KUKA KRL program: MyProgram_203().src

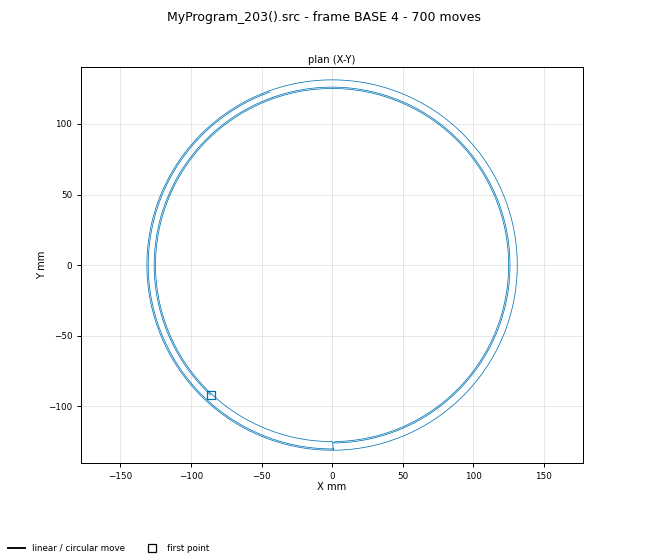
[picture p0: tool path of MyProgram_203().src in frame BASE 4, 700 of 700 moves have a stored position in this frame; points joined in program order, loops and branches not executed]
&ACCESS RVP
&REL 1
&PARAM TEMPLATE = C:\KRC\Roboter\Template\vorgabe
&PARAM EDITMASK = *
DEF MyProgram_203()
; ---- Setting reference (Base) ----
$BASE = BASE_DATA[4]

; --------------------------
; ---- Setting tool (TCP) ----
$TOOL = TOOL_DATA[3]
; --------------------------

$VEL.CP = VEL_APROX_PRINT
Startdeposition()
$VEL.CP = VEL_PRINT
LIN {X -86.0761,Y -92.1467,Z 145,A -135.8963,B 21.9718,C -0.8867,E1 21.8788,E2 583.2193} C_DIS
LIN {X -89.1832,Y -89.1435,Z 145,A -137.9047,B 21.9718,C -0.889,E1 21.8748,E2 585.2313} C_DIS
LIN {X -92.1675,Y -86.0537,Z 145,A -139.8494,B 21.9716,C -0.8935,E1 21.871,E2 587.1736} C_DIS
LIN {X -95.1424,Y -82.7529,Z 145,A -141.8562,B 21.9714,C -0.8986,E1 21.8673,E2 589.1772} C_DIS
LIN {X -97.9193,Y -79.4482,Z 145,A -144.0903,B 21.9716,C -0.8923,E1 21.8633,E2 591.4401} C_DIS
LIN {X -99.986,Y -76.8307,Z 145,A -145.2029,B 21.9709,C -0.9119,E1 21.8615,E2 592.506} C_DIS
LIN {X -101.9983,Y -74.1381,Z 145,A -146.8853,B 21.9709,C -0.9095,E1 21.8587,E2 594.2043} C_DIS
LIN {X -104.8548,Y -70.0396,Z 145,A -149.0462,B 21.9706,C -0.9196,E1 21.8553,E2 596.3505} C_DIS
LIN {X -106.8541,Y -66.9509,Z 145,A -150.8688,B 21.9706,C -0.9179,E1 21.8525,E2 598.1883} C_DIS
LIN {X -109.0384,Y -63.3304,Z 145,A -153.5164,B 21.9715,C -0.8945,E1 21.8487,E2 600.9146} C_DIS
LIN {X -111.7045,Y -58.4954,Z 145,A -154.9531,B 21.9696,C -0.9434,E1 21.847,E2 602.2285} C_DIS
LIN {X -113.7032,Y -54.5088,Z 145,A -157.2159,B 21.9697,C -0.9397,E1 21.8441,E2 604.5155} C_DIS
LIN {X -115.0389,Y -51.6302,Z 145,A -158.7729,B 21.9697,C -0.9392,E1 21.8423,E2 606.0836} C_DIS
LIN {X -116.4531,Y -48.3564,Z 145,A -160.379,B 21.9696,C -0.9444,E1 21.8405,E2 607.686} C_DIS
LIN {X -117.9838,Y -44.4918,Z 145,A -162.2933,B 21.9694,C -0.9489,E1 21.8386,E2 609.6006} C_DIS
LIN {X -119.2139,Y -41.082,Z 145,A -163.8822,B 21.9691,C -0.956,E1 21.8371,E2 611.1808} C_DIS
LIN {X -120.4558,Y -37.2854,Z 145,A -165.5654,B 21.9686,C -0.9666,E1 21.8357,E2 612.8467} C_DIS
LIN {X -121.1863,Y -34.8412,Z 145,A -167.1929,B 21.9692,C -0.9518,E1 21.8344,E2 614.525} C_DIS
LIN {X -122.4757,Y -29.9927,Z 145,A -169.1331,B 21.9684,C -0.9719,E1 21.8331,E2 616.424} C_DIS
LIN {X -123.2253,Y -26.7432,Z 145,A -170.7725,B 21.9684,C -0.9718,E1 21.8321,E2 618.0751} C_DIS
LIN {X -123.9753,Y -23.0268,Z 145,A -172.5489,B 21.9683,C -0.975,E1 21.8311,E2 619.8549} C_DIS
LIN {X -124.6142,Y -19.261,Z 145,A -174.2077,B 21.9679,C -0.9834,E1 21.8304,E2 621.5024} C_DIS
LIN {X -125.1352,Y -15.5323,Z 145,A -176.0548,B 21.9679,C -0.9834,E1 21.8297,E2 623.3622} C_DIS
LIN {X -125.5578,Y -11.6249,Z 145,A -177.7788,B 21.9676,C -0.9915,E1 21.8292,E2 625.0765} C_DIS
LIN {X -125.8536,Y -7.7849,Z 145,A -179.5233,B 21.9673,C -0.9973,E1 21.8289,E2 626.8176} C_DIS
LIN {X -126.0388,Y -3.7439,Z 145,A 178.611,B 21.9671,C -1.002,E1 21.8287,E2 628.6834} C_DIS
LIN {X -126.0974,Y -0.0263,Z 145,A 176.8014,B 21.9671,C -1.0027,E1 21.8287,E2 630.5039} C_DIS
LIN {X -126.0368,Y 3.817,Z 145,A 175.0886,B 21.9668,C -1.0096,E1 21.8287,E2 632.2099} C_DIS
LIN {X -125.8518,Y 7.8139,Z 145,A 173.3197,B 21.9665,C -1.0173,E1 21.829,E2 633.9703} C_DIS
LIN {X -125.5347,Y 11.8647,Z 145,A 171.4401,B 21.9663,C -1.0219,E1 21.8295,E2 635.8506} C_DIS
LIN {X -125.1188,Y 15.6685,Z 145,A 169.6388,B 21.9661,C -1.025,E1 21.83,E2 637.6561} C_DIS
LIN {X -124.595,Y 19.3851,Z 145,A 168.0151,B 21.9657,C -1.0337,E1 21.8307,E2 639.2677} C_DIS
LIN {X -123.9237,Y 23.2965,Z 145,A 165.8228,B 21.9661,C -1.0243,E1 21.8318,E2 641.5001} C_DIS
LIN {X -123.2397,Y 26.6765,Z 145,A 164.7208,B 21.9651,C -1.0473,E1 21.8324,E2 642.5479} C_DIS
LIN {X -122.5731,Y 29.5888,Z 145,A 163.2246,B 21.9651,C -1.0462,E1 21.8334,E2 644.0573} C_DIS
LIN {X -121.6224,Y 33.2883,Z 145,A 161.4104,B 21.9651,C -1.0485,E1 21.8347,E2 645.8773} C_DIS
LIN {X -120.307,Y 37.7657,Z 145,A 159.4485,B 21.9645,C -1.0613,E1 21.8363,E2 647.818} C_DIS
LIN {X -119.4002,Y 40.5435,Z 145,A 158.0205,B 21.9645,C -1.0614,E1 21.8375,E2 649.2549} C_DIS
LIN {X -118.558,Y 42.9378,Z 145,A 156.8422,B 21.9644,C -1.064,E1 21.8386,E2 650.434} C_DIS
LIN {X -117.1974,Y 46.5278,Z 145,A 155.0158,B 21.9643,C -1.0661,E1 21.8405,E2 652.2666} C_DIS
LIN {X -113.3052,Y 55.3334,Z 145,A 150.8392,B 21.9633,C -1.0868,E1 21.8452,E2 656.4139} C_DIS
LIN {X -110.7395,Y 60.3063,Z 145,A 148.2402,B 21.963,C -1.092,E1 21.8486,E2 659.0152} C_DIS
LIN {X -108.9465,Y 63.4891,Z 145,A 146.3727,B 21.9632,C -1.0886,E1 21.8512,E2 660.903} C_DIS
LIN {X -106.7944,Y 67.0458,Z 145,A 144.4384,B 21.963,C -1.0921,E1 21.854,E2 662.8392} C_DIS
LIN {X -104.4846,Y 70.5907,Z 145,A 142.5355,B 21.9628,C -1.0982,E1 21.857,E2 664.7368} C_DIS
LIN {X -102.1644,Y 73.9089,Z 145,A 140.7167,B 21.9625,C -1.104,E1 21.8599,E2 666.5503} C_DIS
LIN {X -99.4483,Y 77.5257,Z 145,A 138.8921,B 21.9618,C -1.1185,E1 21.8629,E2 668.3461} C_DIS
LIN {X -97.8225,Y 79.5671,Z 145,A 137.4168,B 21.9622,C -1.1101,E1 21.8656,E2 669.8517} C_DIS
LIN {X -95.19,Y 82.6983,Z 145,A 135.5368,B 21.962,C -1.114,E1 21.869,E2 671.7312} C_DIS
LIN {X -92.105,Y 86.1209,Z 145,A 133.453,B 21.9617,C -1.1196,E1 21.8729,E2 673.8107} C_DIS
LIN {X -89.2767,Y 89.0495,Z 145,A 131.5891,B 21.9615,C -1.1235,E1 21.8765,E2 675.6733} C_DIS
LIN {X -86.2214,Y 92.0114,Z 145,A 129.6757,B 21.9613,C -1.1287,E1 21.8804,E2 677.5817} C_DIS
LIN {X -83.1134,Y 94.8278,Z 145,A 127.8773,B 21.9609,C -1.1373,E1 21.8841,E2 679.3654} C_DIS
LIN {X -80.3032,Y 97.2188,Z 145,A 126.0625,B 21.9609,C -1.1355,E1 21.888,E2 681.1931} C_DIS
LIN {X -77.0858,Y 99.7893,Z 145,A 124.1693,B 21.9609,C -1.1385,E1 21.8922,E2 683.0862} C_DIS
LIN {X -73.9124,Y 102.1618,Z 145,A 122.2451,B 21.9609,C -1.1373,E1 21.8965,E2 685.0216} C_DIS
LIN {X -70.7167,Y 104.3994,Z 145,A 120.5946,B 21.9605,C -1.1456,E1 21.9003,E2 686.6563} C_DIS
LIN {X -67.5028,Y 106.5059,Z 145,A 118.788,B 21.9605,C -1.1464,E1 21.9045,E2 688.4673} C_DIS
LIN {X -63.9081,Y 108.7007,Z 145,A 116.9174,B 21.9602,C -1.1515,E1 21.909,E2 690.3307} C_DIS
LIN {X -60.038,Y 110.8858,Z 145,A 114.855,B 21.9601,C -1.1532,E1 21.9141,E2 692.3955} C_DIS
LIN {X -56.8206,Y 112.5664,Z 145,A 113.1703,B 21.9601,C -1.1545,E1 21.9182,E2 694.0821} C_DIS
LIN {X -53.2771,Y 114.2861,Z 145,A 111.4983,B 21.9596,C -1.1619,E1 21.9224,E2 695.739} C_DIS
LIN {X -50.183,Y 115.6776,Z 145,A 109.9447,B 21.9596,C -1.1637,E1 21.9264,E2 697.2922} C_DIS
LIN {X -46.4167,Y 117.242,Z 145,A 107.7691,B 21.9601,C -1.1531,E1 21.9321,E2 699.5017} C_DIS
LIN {X -43.3787,Y 118.3991,Z 145,A 106.5136,B 21.9595,C -1.164,E1 21.9353,E2 700.7311} C_DIS
LIN {X -36.9762,Y 120.5504,Z 145,A 103.4705,B 21.9593,C -1.1686,E1 21.9434,E2 703.7683} C_DIS
LIN {X -33.2234,Y 121.6402,Z 145,A 101.5654,B 21.9595,C -1.1651,E1 21.9485,E2 705.6862} C_DIS
LIN {X -29.0003,Y 122.7149,Z 145,A 99.7308,B 21.9591,C -1.1728,E1 21.9535,E2 707.5029} C_DIS
LIN {X -25.2822,Y 123.5334,Z 145,A 98.0319,B 21.9589,C -1.1756,E1 21.9581,E2 709.1969} C_DIS
LIN {X -21.8299,Y 124.1905,Z 145,A 96.3146,B 21.9591,C -1.1718,E1 21.9629,E2 710.9264} C_DIS
LIN {X -17.8466,Y 124.8246,Z 145,A 94.5969,B 21.9588,C -1.1777,E1 21.9676,E2 712.6299} C_DIS
LIN {X -14.2799,Y 125.2846,Z 145,A 92.9165,B 21.9588,C -1.1767,E1 21.9722,E2 714.3144} C_DIS
LIN {X -10.3602,Y 125.668,Z 145,A 91.0232,B 21.9591,C -1.1732,E1 21.9775,E2 716.2181} C_DIS
LIN {X -5.674,Y 125.968,Z 145,A 88.9107,B 21.959,C -1.1748,E1 21.9834,E2 718.327} C_DIS
LIN {X -1.8806,Y 126.0803,Z 145,A 87.2175,B 21.9589,C -1.1765,E1 21.9881,E2 720.0158} C_DIS
LIN {X 2.6511,Y 126.0675,Z 145,A 85.1051,B 21.9589,C -1.1745,E1 21.994,E2 722.1331} C_DIS
LIN {X 6.9515,Y 125.9039,Z 145,A 83.2593,B 21.9588,C -1.1791,E1 21.9991,E2 723.966} C_DIS
LIN {X 10.5423,Y 125.6526,Z 145,A 81.648,B 21.9588,C -1.1801,E1 22.0036,E2 725.5738} C_DIS
LIN {X 14.0573,Y 125.3093,Z 145,A 79.8978,B 21.959,C -1.1736,E1 22.0085,E2 727.3398} C_DIS
LIN {X 18.2331,Y 124.7694,Z 145,A 78.1356,B 21.9587,C -1.1795,E1 22.0133,E2 729.0846} C_DIS
LIN {X 22.0415,Y 124.1527,Z 145,A 76.3822,B 21.9587,C -1.1789,E1 22.0182,E2 730.8376} C_DIS
LIN {X 25.7971,Y 123.4286,Z 145,A 74.5556,B 21.959,C -1.1743,E1 22.0232,E2 732.6739} C_DIS
LIN {X 29.4691,Y 122.6019,Z 145,A 72.9585,B 21.9588,C -1.1782,E1 22.0275,E2 734.2581} C_DIS
LIN {X 32.7186,Y 121.7752,Z 145,A 71.476,B 21.9588,C -1.1789,E1 22.0315,E2 735.7358} C_DIS
LIN {X 36.0284,Y 120.8387,Z 145,A 69.5967,B 21.9595,C -1.1642,E1 22.0366,E2 737.6507} C_DIS
LIN {X 40.2853,Y 119.4862,Z 145,A 67.8211,B 21.9591,C -1.1734,E1 22.0413,E2 739.3978} C_DIS
LIN {X 44.8165,Y 117.8622,Z 145,A 65.6246,B 21.9591,C -1.171,E1 22.047,E2 741.5956} C_DIS
LIN {X 48.3157,Y 116.4701,Z 145,A 63.9039,B 21.9593,C -1.1688,E1 22.0515,E2 743.3176} C_DIS
LIN {X 51.3332,Y 115.1717,Z 145,A 62.4227,B 21.9593,C -1.1676,E1 22.0553,E2 744.7977} C_DIS
LIN {X 54.3914,Y 113.7593,Z 145,A 60.934,B 21.9593,C -1.1676,E1 22.059,E2 746.2821} C_DIS
LIN {X 57.5159,Y 112.2125,Z 145,A 59.2771,B 21.9596,C -1.1624,E1 22.0632,E2 747.9476} C_DIS
LIN {X 61.6301,Y 110.0083,Z 145,A 57.1457,B 21.9598,C -1.159,E1 22.0684,E2 750.0811} C_DIS
LIN {X 65.4184,Y 107.7987,Z 145,A 55.2232,B 21.9598,C -1.159,E1 22.073,E2 751.9964} C_DIS
LIN {X 68.8019,Y 105.6712,Z 145,A 52.7949,B 21.9612,C -1.1295,E1 22.0789,E2 754.4942} C_DIS
LIN {X 72.8559,Y 102.9174,Z 145,A 51.3065,B 21.9598,C -1.158,E1 22.0821,E2 755.9008} C_DIS
LIN {X 75.3902,Y 101.0762,Z 145,A 49.7164,B 21.9603,C -1.1482,E1 22.0857,E2 757.5106} C_DIS
LIN {X 78.8216,Y 98.4244,Z 145,A 47.7508,B 21.9605,C -1.1448,E1 22.09,E2 759.4768} C_DIS
LIN {X 82.0406,Y 95.7576,Z 145,A 45.8388,B 21.9607,C -1.1405,E1 22.0941,E2 761.3916} C_DIS
LIN {X 85.4008,Y 92.7728,Z 145,A 43.8587,B 21.9607,C -1.1392,E1 22.0982,E2 763.3661} C_DIS
LIN {X 88.4403,Y 89.88,Z 145,A 41.9475,B 21.961,C -1.135,E1 22.102,E2 765.2792} C_DIS
LIN {X 91.391,Y 86.8785,Z 145,A 40.0249,B 21.9612,C -1.1304,E1 22.1058,E2 767.2045} C_DIS
LIN {X 93.6073,Y 84.4858,Z 145,A 38.5847,B 21.9612,C -1.1289,E1 22.1085,E2 768.6413} C_DIS
LIN {X 96.3788,Y 81.31,Z 145,A 36.0715,B 21.9628,C -1.0979,E1 22.1132,E2 771.2237} C_DIS
LIN {X 99.535,Y 77.4131,Z 145,A 34.5935,B 21.9613,C -1.1281,E1 22.1156,E2 772.6133} C_DIS
LIN {X 101.1414,Y 75.3027,Z 145,A 33.1546,B 21.962,C -1.1147,E1 22.118,E2 774.0801} C_DIS
LIN {X 103.7943,Y 71.6024,Z 145,A 31.1509,B 21.962,C -1.1124,E1 22.1212,E2 776.0786} C_DIS
LIN {X 106.1382,Y 68.0791,Z 145,A 29.1772,B 21.9624,C -1.1052,E1 22.1242,E2 778.0601} C_DIS
LIN {X 108.4285,Y 64.3692,Z 145,A 27.304,B 21.9624,C -1.1048,E1 22.1269,E2 779.9233} C_DIS
LIN {X 110.3157,Y 61.0781,Z 145,A 25.7873,B 21.9622,C -1.1095,E1 22.129,E2 781.4184} C_DIS
LIN {X 111.6871,Y 58.5286,Z 145,A 24.3527,B 21.9626,C -1.1006,E1 22.1309,E2 782.868} C_DIS
LIN {X 113.193,Y 55.5608,Z 145,A 22.834,B 21.9629,C -1.0961,E1 22.1328,E2 784.3893} C_DIS
LIN {X 114.5601,Y 52.6845,Z 145,A 21.3651,B 21.9631,C -1.091,E1 22.1345,E2 785.8626} C_DIS
LIN {X 117.083,Y 46.8114,Z 145,A 18.5463,B 21.9633,C -1.0865,E1 22.1376,E2 788.6754} C_DIS
LIN {X 118.1916,Y 43.937,Z 145,A 17.1359,B 21.9635,C -1.0819,E1 22.139,E2 790.0889} C_DIS
LIN {X 119.3991,Y 40.5467,Z 145,A 15.2634,B 21.9642,C -1.0663,E1 22.1407,E2 791.9907} C_DIS
LIN {X 120.5527,Y 36.9689,Z 145,A 13.7751,B 21.964,C -1.0712,E1 22.142,E2 793.4562} C_DIS
LIN {X 121.6013,Y 33.3639,Z 145,A 12.0113,B 21.9644,C -1.0634,E1 22.1433,E2 795.2292} C_DIS
LIN {X 122.5655,Y 29.6202,Z 145,A 10.3631,B 21.9644,C -1.063,E1 22.1444,E2 796.8674} C_DIS
LIN {X 123.3293,Y 26.2616,Z 145,A 8.698,B 21.9648,C -1.0536,E1 22.1454,E2 798.5463} C_DIS
LIN {X 124.1128,Y 22.264,Z 145,A 6.9712,B 21.9648,C -1.0536,E1 22.1463,E2 800.2616} C_DIS
LIN {X 124.6972,Y 18.7236,Z 145,A 5.3351,B 21.9651,C -1.0482,E1 22.147,E2 801.9009} C_DIS
LIN {X 125.181,Y 15.1483,Z 145,A 3.697,B 21.9653,C -1.0431,E1 22.1476,E2 803.5414} C_DIS
LIN {X 125.5665,Y 11.5343,Z 145,A 1.8734,B 21.9659,C -1.03,E1 22.1481,E2 805.3873} C_DIS
LIN {X 125.8923,Y 7.1553,Z 145,A -0.0848,B 21.9661,C -1.0253,E1 22.1485,E2 807.3445} C_DIS
LIN {X 126.0698,Y 2.5107,Z 145,A -2.008,B 21.9661,C -1.0272,E1 22.1486,E2 809.2494} C_DIS
LIN {X 126.0934,Y -0.7076,Z 145,A -3.5783,B 21.9664,C -1.0176,E1 22.1486,E2 810.8345} C_DIS
LIN {X 126.0148,Y -4.4933,Z 145,A -4.9898,B 21.9661,C -1.0263,E1 22.1486,E2 812.2131} C_DIS
LIN {X 125.8818,Y -7.3261,Z 145,A -6.4589,B 21.9666,C -1.0139,E1 22.1483,E2 813.7052} C_DIS
LIN {X 125.6288,Y -10.8246,Z 145,A -7.9964,B 21.9667,C -1.0114,E1 22.148,E2 815.2388} C_DIS
LIN {X 125.2804,Y -14.3147,Z 145,A -9.8028,B 21.9674,C -0.9965,E1 22.1474,E2 817.0724} C_DIS
LIN {X 124.5584,Y -19.6216,Z 145,A -11.9587,B 21.9671,C -1.0015,E1 22.1466,E2 819.2004} C_DIS
LIN {X 123.9753,Y -23.0268,Z 145,A -13.6498,B 21.9676,C -0.9909,E1 22.1457,E2 820.9081} C_DIS
LIN {X 123.2202,Y -26.7671,Z 145,A -15.2366,B 21.9676,C -0.9922,E1 22.1448,E2 822.4809} C_DIS
LIN {X 122.5183,Y -29.816,Z 145,A -16.6631,B 21.9678,C -0.9875,E1 22.1439,E2 823.9104} C_DIS
LIN {X 121.587,Y -33.415,Z 145,A -19.208,B 21.9696,C -0.9431,E1 22.142,E2 826.556} C_DIS
LIN {X 119.9115,Y -39.004,Z 145,A -21.2058,B 21.9687,C -0.9646,E1 22.1403,E2 828.4838} C_DIS
LIN {X 118.522,Y -43.0377,Z 145,A -22.8902,B 21.9685,C -0.9703,E1 22.1388,E2 830.1421} C_DIS
LIN {X 117.3012,Y -46.2648,Z 145,A -24.4554,B 21.9687,C -0.9656,E1 22.1372,E2 831.7098} C_DIS
LIN {X 116.0348,Y -49.3567,Z 145,A -26.2843,B 21.9695,C -0.9468,E1 22.1352,E2 833.5771} C_DIS
LIN {X 114.192,Y -53.4805,Z 145,A -27.9918,B 21.9691,C -0.9564,E1 22.1332,E2 835.2483} C_DIS
LIN {X 112.9996,Y -55.9528,Z 145,A -29.2419,B 21.9692,C -0.9526,E1 22.1317,E2 836.5007} C_DIS
LIN {X 111.5677,Y -58.7559,Z 145,A -30.6943,B 21.9694,C -0.9474,E1 22.1298,E2 837.9581} C_DIS
LIN {X 109.6782,Y -62.2162,Z 145,A -32.5002,B 21.9697,C -0.9416,E1 22.1274,E2 839.7688} C_DIS
LIN {X 107.8477,Y -65.3372,Z 145,A -34.238,B 21.97,C -0.9326,E1 22.1249,E2 841.5201} C_DIS
LIN {X 104.5043,Y -70.5616,Z 145,A -36.9004,B 21.97,C -0.9318,E1 22.1208,E2 844.1691} C_DIS
LIN {X 102.302,Y -73.7189,Z 145,A -38.6817,B 21.9703,C -0.9256,E1 22.1179,E2 845.9569} C_DIS
LIN {X 98.1665,Y -79.1418,Z 145,A -41.554,B 21.9703,C -0.9277,E1 22.1131,E2 848.808} C_DIS
LIN {X 96.4896,Y -81.1779,Z 145,A -43.3712,B 21.9715,C -0.8966,E1 22.1097,E2 850.6984} C_DIS
LIN {X 93.891,Y -84.1698,Z 145,A -44.4741,B 21.9704,C -0.9236,E1 22.1078,E2 851.7237} C_DIS
LIN {X 91.0602,Y -87.2237,Z 145,A -46.7454,B 21.9713,C -0.9017,E1 22.1034,E2 854.0417} C_DIS
LIN {X 85.1894,Y -92.9671,Z 145,A -50.1898,B 21.9711,C -0.9058,E1 22.0965,E2 857.4586} C_DIS
LIN {X 79.9571,Y -97.5038,Z 145,A -53.6103,B 21.9718,C -0.8865,E1 22.0892,E2 860.9153} C_DIS
LIN {X 76.2357,Y -100.4406,Z 145,A -55.6577,B 21.9718,C -0.8867,E1 22.0847,E2 862.9534} C_DIS
LIN {X 72.0753,Y -103.4661,Z 145,A -57.7745,B 21.9716,C -0.8918,E1 22.0799,E2 865.0479} C_DIS
LIN {X 70.1868,Y -104.7565,Z 145,A -59.0333,B 21.9721,C -0.88,E1 22.0769,E2 866.3334} C_DIS
LIN {X 66.3539,Y -107.2256,Z 145,A -60.9981,B 21.9721,C -0.8808,E1 22.0723,E2 868.2885} C_DIS
LIN {X 62.8473,Y -109.3179,Z 145,A -62.9619,B 21.9724,C -0.8727,E1 22.0676,E2 870.2672} C_DIS
LIN {X 58.542,Y -111.6801,Z 145,A -65.0598,B 21.9723,C -0.8749,E1 22.0624,E2 872.3523} C_DIS
LIN {X 55.5659,Y -113.1905,Z 145,A -66.5844,B 21.9723,C -0.8721,E1 22.0586,E2 873.8797} C_DIS
LIN {X 49.5781,Y -115.9391,Z 145,A -69.4969,B 21.9724,C -0.8711,E1 22.0512,E2 876.7863} C_DIS
LIN {X 46.7448,Y -117.1099,Z 145,A -70.9423,B 21.9726,C -0.8669,E1 22.0475,E2 878.2391} C_DIS
LIN {X 41.7584,Y -118.9794,Z 145,A -73.7577,B 21.9733,C -0.8464,E1 22.04,E2 881.1025} C_DIS
LIN {X 38.3256,Y -120.1282,Z 145,A -75.0565,B 21.9729,C -0.8596,E1 22.0366,E2 882.3632} C_DIS
LIN {X 34.3264,Y -121.3321,Z 145,A -76.9584,B 21.9729,C -0.8573,E1 22.0315,E2 884.2674} C_DIS
LIN {X 30.6828,Y -122.3043,Z 145,A -78.7231,B 21.9731,C -0.8534,E1 22.0267,E2 886.0395} C_DIS
LIN {X 26.5483,Y -123.2674,Z 145,A -80.5362,B 21.973,C -0.8567,E1 22.0218,E2 887.8409} C_DIS
LIN {X 22.8688,Y -124.0046,Z 145,A -82.3187,B 21.9731,C -0.8519,E1 22.0169,E2 889.6337} C_DIS
LIN {X 17.2731,Y -124.9066,Z 145,A -84.6046,B 21.9727,C -0.8627,E1 22.0107,E2 891.8883} C_DIS
LIN {X 13.2738,Y -125.3936,Z 145,A -86.5916,B 21.973,C -0.8549,E1 22.0051,E2 893.8944} C_DIS
LIN {X 10.0614,Y -125.6932,Z 145,A -88.3078,B 21.9735,C -0.8434,E1 22.0002,E2 895.6404} C_DIS
LIN {X 4.1739,Y -126.0268,Z 145,A -90.6923,B 21.973,C -0.8551,E1 21.9937,E2 897.9926} C_DIS
LIN {X 0.8946,Y -126.0892,Z 145,A -92.1733,B 21.973,C -0.8551,E1 21.9895,E2 899.4731} C_DIS
Enddeposition()
LIN {X 0.8946,Y -126.0892,Z 145,A -92.1733,B 21.973,C -0.8551,E1 21.9895,E2 899.4731} C_DIS
Startdeposition()
$VEL.CP = VEL_PRINT
LIN {X 2.2905,Y -125.1132,Z 145,A -90.6676,B 20.9492,C -0.7352,E1 20.9658,E2 898.1754} C_DIS
LIN {X 5.3456,Y -125.0206,Z 145,A -89.2758,B 20.9492,C -0.7352,E1 20.9697,E2 896.7837} C_DIS
LIN {X 8.3882,Y -124.8543,Z 145,A -87.8298,B 20.9492,C -0.7379,E1 20.9737,E2 895.331} C_DIS
LIN {X 12.2611,Y -124.5321,Z 145,A -85.9295,B 20.9489,C -0.7438,E1 20.9791,E2 893.4156} C_DIS
LIN {X 16.0664,Y -124.0982,Z 145,A -84.334,B 20.9491,C -0.7383,E1 20.9834,E2 891.8371} C_DIS
LIN {X 19.1002,Y -123.6675,Z 145,A -82.9291,B 20.9491,C -0.7393,E1 20.9873,E2 890.431} C_DIS
LIN {X 22.1459,Y -123.1585,Z 145,A -81.5254,B 20.9491,C -0.7399,E1 20.9912,E2 889.0273} C_DIS
LIN {X 25.1624,Y -122.5779,Z 145,A -80.1227,B 20.9491,C -0.7409,E1 20.995,E2 887.624} C_DIS
LIN {X 28.1526,Y -121.926,Z 145,A -78.7132,B 20.9489,C -0.7425,E1 20.9989,E2 886.2124} C_DIS
LIN {X 31.9271,Y -120.9925,Z 145,A -76.8026,B 20.9487,C -0.7497,E1 21.0041,E2 884.2852} C_DIS
LIN {X 35.5906,Y -119.9663,Z 145,A -75.2093,B 20.9489,C -0.7453,E1 21.0083,E2 882.7075} C_DIS
LIN {X 39.227,Y -118.8265,Z 145,A -73.3406,B 20.9486,C -0.7525,E1 21.0133,E2 880.8228} C_DIS
LIN {X 43.1623,Y -117.4563,Z 145,A -71.421,B 20.9486,C -0.7554,E1 21.0184,E2 878.9} C_DIS
LIN {X 46.4597,Y -116.1895,Z 145,A -69.8013,B 20.9484,C -0.7577,E1 21.0226,E2 877.2783} C_DIS
LIN {X 50.6906,Y -114.4073,Z 145,A -67.8654,B 20.9486,C -0.7536,E1 21.0275,E2 875.3594} C_DIS
LIN {X 53.4692,Y -113.1357,Z 145,A -66.3999,B 20.9484,C -0.7586,E1 21.0313,E2 873.8847} C_DIS
LIN {X 56.2603,Y -111.7742,Z 145,A -65.0568,B 20.9484,C -0.7575,E1 21.0346,E2 872.549} C_DIS
LIN {X 59.5508,Y -110.0576,Z 145,A -63.326,B 20.9483,C -0.7616,E1 21.0389,E2 870.8127} C_DIS
LIN {X 63.0135,Y -108.1123,Z 145,A -61.3844,B 20.948,C -0.77,E1 21.0436,E2 868.8546} C_DIS
LIN {X 66.9426,Y -105.724,Z 145,A -59.2931,B 20.9479,C -0.7733,E1 21.0486,E2 866.7623} C_DIS
LIN {X 70.7812,Y -103.1933,Z 145,A -57.1931,B 20.9477,C -0.7771,E1 21.0535,E2 864.6603} C_DIS
LIN {X 74.5429,Y -100.51,Z 145,A -55.1021,B 20.9477,C -0.7804,E1 21.0582,E2 862.5694} C_DIS
LIN {X 78.175,Y -97.7118,Z 145,A -53.0797,B 20.9476,C -0.7815,E1 21.0626,E2 860.5529} C_DIS
LIN {X 81.4027,Y -95.0398,Z 145,A -51.0996,B 20.9473,C -0.7883,E1 21.0669,E2 858.5631} C_DIS
LIN {X 84.596,Y -92.2083,Z 145,A -49.2391,B 20.9473,C -0.7887,E1 21.0707,E2 856.7107} C_DIS
LIN {X 87.3367,Y -89.6175,Z 145,A -47.4398,B 20.9471,C -0.7959,E1 21.0743,E2 854.9005} C_DIS
LIN {X 90.416,Y -86.509,Z 145,A -45.6663,B 20.9473,C -0.7907,E1 21.0778,E2 853.1506} C_DIS
LIN {X 92.7211,Y -84.0336,Z 145,A -44.0016,B 20.9469,C -0.7995,E1 21.0809,E2 851.4702} C_DIS
LIN {X 95.4663,Y -80.9015,Z 145,A -42.1049,B 20.9468,C -0.8039,E1 21.0844,E2 849.5719} C_DIS
LIN {X 98.076,Y -77.7176,Z 145,A -40.1671,B 20.9465,C -0.8111,E1 21.0878,E2 847.625} C_DIS
LIN {X 100.5105,Y -74.5421,Z 145,A -38.3169,B 20.9463,C -0.8167,E1 21.0909,E2 845.7699} C_DIS
LIN {X 103.1762,Y -70.8062,Z 145,A -36.2351,B 20.9461,C -0.8215,E1 21.0943,E2 843.6872} C_DIS
LIN {X 105.7003,Y -66.9802,Z 145,A -34.2557,B 20.9461,C -0.8221,E1 21.0972,E2 841.7183} C_DIS
LIN {X 107.723,Y -63.6766,Z 145,A -32.3868,B 20.9458,C -0.8312,E1 21.0999,E2 839.8356} C_DIS
LIN {X 109.9886,Y -59.6776,Z 145,A -30.3807,B 20.9457,C -0.8329,E1 21.1027,E2 837.8374} C_DIS
LIN {X 111.5783,Y -56.645,Z 145,A -28.9441,B 20.9457,C -0.8318,E1 21.1045,E2 836.4134} C_DIS
LIN {X 113.1197,Y -53.5027,Z 145,A -27.1385,B 20.9452,C -0.8454,E1 21.1067,E2 834.5817} C_DIS
LIN {X 114.7157,Y -49.9882,Z 145,A -25.3977,B 20.9451,C -0.8495,E1 21.1087,E2 832.8411} C_DIS
LIN {X 116.4728,Y -45.7456,Z 145,A -23.4688,B 20.9451,C -0.8481,E1 21.1107,E2 830.9288} C_DIS
LIN {X 117.5553,Y -42.8878,Z 145,A -22.0755,B 20.945,C -0.8521,E1 21.112,E2 829.534} C_DIS
LIN {X 118.5803,Y -39.9665,Z 145,A -20.5052,B 20.9445,C -0.8632,E1 21.1135,E2 827.9437} C_DIS
LIN {X 119.9568,Y -35.6232,Z 145,A -18.5999,B 20.9445,C -0.8616,E1 21.115,E2 826.0559} C_DIS
LIN {X 120.9804,Y -31.9723,Z 145,A -16.8665,B 20.9444,C -0.8669,E1 21.1163,E2 824.32} C_DIS
LIN {X 121.7499,Y -28.9061,Z 145,A -15.4436,B 20.9442,C -0.8703,E1 21.1172,E2 822.8976} C_DIS
LIN {X 122.4223,Y -25.9129,Z 145,A -14.052,B 20.9441,C -0.8741,E1 21.1181,E2 821.5052} C_DIS
LIN {X 123.0211,Y -22.9043,Z 145,A -12.6367,B 20.9439,C -0.879,E1 21.1188,E2 820.0864} C_DIS
LIN {X 123.5463,Y -19.8818,Z 145,A -11.2496,B 20.9438,C -0.8826,E1 21.1194,E2 818.6991} C_DIS
LIN {X 123.9959,Y -16.8474,Z 145,A -9.8472,B 20.9436,C -0.887,E1 21.12,E2 817.2946} C_DIS
LIN {X 124.455,Y -13.0216,Z 145,A -8.1253,B 20.9434,C -0.8907,E1 21.1205,E2 815.5748} C_DIS
LIN {X 124.7494,Y -9.8273,Z 145,A -6.6794,B 20.9433,C -0.8943,E1 21.1209,E2 814.1293} C_DIS
LIN {X 124.9441,Y -6.9191,Z 145,A -5.3144,B 20.9431,C -0.8999,E1 21.1211,E2 812.7586} C_DIS
LIN {X 125.0965,Y -3.0838,Z 145,A -3.6051,B 20.9429,C -0.9034,E1 21.1213,E2 811.052} C_DIS
LIN {X 125.1348,Y 0.42,Z 145,A -1.8881,B 20.9425,C -0.9134,E1 21.1213,E2 809.3196} C_DIS
LIN {X 125.0758,Y 3.8284,Z 145,A -0.4626,B 20.9425,C -0.9124,E1 21.1212,E2 807.9072} C_DIS
LIN {X 124.9445,Y 6.9116,Z 145,A 0.9446,B 20.9424,C -0.9166,E1 21.121,E2 806.4986} C_DIS
LIN {X 124.7049,Y 10.353,Z 145,A 2.5934,B 20.942,C -0.9246,E1 21.1206,E2 804.8394} C_DIS
LIN {X 124.372,Y 13.7929,Z 145,A 4.0803,B 20.942,C -0.9253,E1 21.1202,E2 803.3611} C_DIS
LIN {X 123.9973,Y 16.8364,Z 145,A 5.4714,B 20.9418,C -0.9291,E1 21.1197,E2 801.9694} C_DIS
LIN {X 123.5461,Y 19.8831,Z 145,A 7.0413,B 20.9413,C -0.9405,E1 21.119,E2 800.3792} C_DIS
LIN {X 122.8768,Y 23.6594,Z 145,A 8.6246,B 20.9414,C -0.9384,E1 21.1182,E2 798.8132} C_DIS
LIN {X 122.259,Y 26.6689,Z 145,A 10.0185,B 20.9413,C -0.9421,E1 21.1174,E2 797.4187} C_DIS
LIN {X 121.3841,Y 30.4052,Z 145,A 11.8297,B 20.9409,C -0.9498,E1 21.1162,E2 795.5988} C_DIS
LIN {X 120.3946,Y 34.1135,Z 145,A 13.6748,B 20.9406,C -0.9589,E1 21.1149,E2 793.7412} C_DIS
LIN {X 119.2551,Y 37.9033,Z 145,A 15.4255,B 20.9404,C -0.9616,E1 21.1134,E2 791.9951} C_DIS
LIN {X 117.9198,Y 41.8767,Z 145,A 17.3039,B 20.9403,C -0.9655,E1 21.1117,E2 790.119} C_DIS
LIN {X 116.4765,Y 45.736,Z 145,A 19.2476,B 20.9399,C -0.9734,E1 21.1097,E2 788.1663} C_DIS
LIN {X 114.7074,Y 50.0073,Z 145,A 21.3411,B 20.9397,C -0.9784,E1 21.1075,E2 786.0728} C_DIS
LIN {X 113.1199,Y 53.5024,Z 145,A 22.9291,B 20.9398,C -0.9759,E1 21.1056,E2 784.5022} C_DIS
LIN {X 111.7752,Y 56.2583,Z 145,A 24.3215,B 20.9397,C -0.9793,E1 21.1039,E2 783.1095} C_DIS
LIN {X 110.0408,Y 59.582,Z 145,A 26.0594,B 20.9394,C -0.9849,E1 21.1016,E2 781.3673} C_DIS
LIN {X 108.1119,Y 63.0143,Z 145,A 27.9861,B 20.9389,C -0.995,E1 21.0989,E2 779.4244} C_DIS
LIN {X 105.7204,Y 66.9483,Z 145,A 30.0777,B 20.9387,C -0.9998,E1 21.0958,E2 777.3325} C_DIS
LIN {X 103.1871,Y 70.7902,Z 145,A 32.1684,B 20.9385,C -1.0044,E1 21.0926,E2 775.2415} C_DIS
LIN {X 100.4979,Y 74.5592,Z 145,A 34.2558,B 20.9383,C -1.0082,E1 21.0891,E2 773.1558} C_DIS
LIN {X 97.7656,Y 78.1075,Z 145,A 36.2899,B 20.9381,C -1.0124,E1 21.0856,E2 771.1216} C_DIS
LIN {X 94.949,Y 81.508,Z 145,A 38.2974,B 20.938,C -1.0165,E1 21.082,E2 769.114} C_DIS
LIN {X 91.936,Y 84.8922,Z 145,A 40.3126,B 20.9379,C -1.0186,E1 21.0782,E2 767.1039} C_DIS
LIN {X 89.0241,Y 87.9413,Z 145,A 42.3108,B 20.9375,C -1.0256,E1 21.0743,E2 765.0966} C_DIS
LIN {X 86.0103,Y 90.8906,Z 145,A 44.1533,B 20.9375,C -1.0258,E1 21.0706,E2 763.2627} C_DIS
LIN {X 83.0295,Y 93.6215,Z 145,A 46.0479,B 20.9373,C -1.0314,E1 21.0667,E2 761.3619} C_DIS
LIN {X 79.6781,Y 96.4897,Z 145,A 47.9933,B 20.9373,C -1.0321,E1 21.0626,E2 759.4237} C_DIS
LIN {X 76.3839,Y 99.1184,Z 145,A 50.0112,B 20.9369,C -1.0393,E1 21.0581,E2 757.3947} C_DIS
LIN {X 72.7531,Y 101.8127,Z 145,A 52.0397,B 20.9369,C -1.0412,E1 21.0535,E2 755.3698} C_DIS
LIN {X 69.2291,Y 104.2414,Z 145,A 53.9511,B 20.9367,C -1.0423,E1 21.0491,E2 753.463} C_DIS
LIN {X 66.3019,Y 106.127,Z 145,A 55.602,B 20.9365,C -1.0472,E1 21.0452,E2 751.8051} C_DIS
LIN {X 62.3472,Y 108.498,Z 145,A 57.7106,B 20.9364,C -1.0502,E1 21.0401,E2 749.6961} C_DIS
LIN {X 58.4796,Y 110.6283,Z 145,A 59.6149,B 20.9364,C -1.048,E1 21.0355,E2 747.8043} C_DIS
LIN {X 55.5671,Y 112.1192,Z 145,A 61.0533,B 20.9365,C -1.0475,E1 21.0319,E2 746.3722} C_DIS
LIN {X 52.8029,Y 113.4474,Z 145,A 62.4546,B 20.9365,C -1.049,E1 21.0284,E2 744.971} C_DIS
LIN {X 49.3041,Y 115.0114,Z 145,A 64.3604,B 20.936,C -1.0573,E1 21.0234,E2 743.0479} C_DIS
LIN {X 45.7559,Y 116.4688,Z 145,A 65.9554,B 20.9363,C -1.0524,E1 21.0194,E2 741.4709} C_DIS
LIN {X 42.859,Y 117.5657,Z 145,A 67.368,B 20.9363,C -1.0535,E1 21.0157,E2 740.0588} C_DIS
LIN {X 39.9845,Y 118.5743,Z 145,A 68.7648,B 20.9361,C -1.0548,E1 21.012,E2 738.6618} C_DIS
LIN {X 36.6634,Y 119.642,Z 145,A 70.4221,B 20.936,C -1.0586,E1 21.0075,E2 736.9977} C_DIS
LIN {X 32.6355,Y 120.8036,Z 145,A 72.4358,B 20.9357,C -1.0638,E1 21.0021,E2 734.9735} C_DIS
LIN {X 28.1804,Y 121.9196,Z 145,A 74.3849,B 20.936,C -1.0587,E1 20.9969,E2 733.0419} C_DIS
LIN {X 25.1648,Y 122.5774,Z 145,A 75.7915,B 20.936,C -1.0591,E1 20.993,E2 731.6363} C_DIS
LIN {X 22.1493,Y 123.1579,Z 145,A 77.1924,B 20.936,C -1.0595,E1 20.9892,E2 730.2362} C_DIS
LIN {X 19.1296,Y 123.6629,Z 145,A 78.593,B 20.9359,C -1.06,E1 20.9853,E2 728.8361} C_DIS
LIN {X 16.094,Y 124.0946,Z 145,A 80.012,B 20.9359,C -1.061,E1 20.9814,E2 727.4158} C_DIS
LIN {X 12.2653,Y 124.5317,Z 145,A 81.8976,B 20.9356,C -1.0662,E1 20.9761,E2 725.5172} C_DIS
LIN {X 8.3378,Y 124.8575,Z 145,A 83.5411,B 20.9359,C -1.0598,E1 20.9716,E2 723.8925} C_DIS
LIN {X 4.9384,Y 125.0364,Z 145,A 85.1733,B 20.9358,C -1.0628,E1 20.967,E2 722.2527} C_DIS
LIN {X 1.065,Y 125.13,Z 145,A 86.9736,B 20.9358,C -1.0636,E1 20.962,E2 720.4502} C_DIS
LIN {X -2.3023,Y 125.113,Z 145,A 88.5309,B 20.9358,C -1.0639,E1 20.9576,E2 718.892} C_DIS
LIN {X -6.1306,Y 124.9837,Z 145,A 90.199,B 20.9358,C -1.06,E1 20.953,E2 717.2345} C_DIS
LIN {X -9.1901,Y 124.796,Z 145,A 91.5968,B 20.9359,C -1.0593,E1 20.9491,E2 715.8381} C_DIS
LIN {X -12.266,Y 124.5316,Z 145,A 93.0069,B 20.9359,C -1.0585,E1 20.9452,E2 714.4294} C_DIS
LIN {X -15.3141,Y 124.1942,Z 145,A 94.4098,B 20.936,C -1.0577,E1 20.9413,E2 713.0275} C_DIS
LIN {X -18.619,Y 123.7419,Z 145,A 95.8553,B 20.9362,C -1.0536,E1 20.9373,E2 711.5922} C_DIS
LIN {X -21.8235,Y 123.2162,Z 145,A 97.4743,B 20.936,C -1.0578,E1 20.9328,E2 709.9596} C_DIS
LIN {X -25.1671,Y 122.5769,Z 145,A 98.9999,B 20.9361,C -1.0553,E1 20.9287,E2 708.4389} C_DIS
LIN {X -28.1578,Y 121.9248,Z 145,A 100.5609,B 20.9359,C -1.0604,E1 20.9244,E2 706.8613} C_DIS
LIN {X -32.6668,Y 120.7952,Z 145,A 102.6998,B 20.9359,C -1.0587,E1 20.9186,E2 704.7231} C_DIS
LIN {X -37.011,Y 119.5356,Z 145,A 104.772,B 20.9361,C -1.0566,E1 20.9131,E2 702.6526} C_DIS
LIN {X -41.2133,Y 118.1521,Z 145,A 106.6783,B 20.9364,C -1.0496,E1 20.9081,E2 700.7616} C_DIS
LIN {X -45.0232,Y 116.7536,Z 145,A 108.5164,B 20.9365,C -1.0465,E1 20.9033,E2 698.9276} C_DIS
LIN {X -48.5945,Y 115.3131,Z 145,A 110.439,B 20.9364,C -1.0503,E1 20.8983,E2 696.9891} C_DIS
LIN {X -52.1017,Y 113.7717,Z 145,A 112.038,B 20.9368,C -1.0418,E1 20.8942,E2 695.4093} C_DIS
LIN {X -54.8726,Y 112.4618,Z 145,A 113.4449,B 20.9368,C -1.0398,E1 20.8907,E2 694.0036} C_DIS
LIN {X -57.9544,Y 110.904,Z 145,A 115.0725,B 20.9368,C -1.0391,E1 20.8866,E2 692.3726} C_DIS
LIN {X -61.6844,Y 108.8761,Z 145,A 117.1523,B 20.9368,C -1.041,E1 20.8815,E2 690.28} C_DIS
LIN {X -65.6444,Y 106.5351,Z 145,A 119.2753,B 20.937,C -1.0379,E1 20.8765,E2 688.1578} C_DIS
LIN {X -69.5186,Y 104.0481,Z 145,A 121.382,B 20.9371,C -1.034,E1 20.8716,E2 686.0538} C_DIS
LIN {X -72.6901,Y 101.8578,Z 145,A 123.1522,B 20.9373,C -1.0307,E1 20.8675,E2 684.2853} C_DIS
LIN {X -76.3798,Y 99.1216,Z 145,A 125.2726,B 20.9375,C -1.0271,E1 20.8628,E2 682.1658} C_DIS
LIN {X -79.6733,Y 96.4937,Z 145,A 127.1334,B 20.9378,C -1.0204,E1 20.8588,E2 680.3152} C_DIS
LIN {X -82.589,Y 94.0109,Z 145,A 128.9839,B 20.9378,C -1.0203,E1 20.8549,E2 678.4564} C_DIS
LIN {X -85.727,Y 91.1579,Z 145,A 130.8502,B 20.9381,C -1.013,E1 20.8511,E2 676.6012} C_DIS
LIN {X -88.4765,Y 88.4923,Z 145,A 132.6983,B 20.9381,C -1.0125,E1 20.8474,E2 674.7452} C_DIS
LIN {X -91.4022,Y 85.4666,Z 145,A 134.5632,B 20.9385,C -1.0055,E1 20.8438,E2 672.8899} C_DIS
LIN {X -93.9979,Y 82.6037,Z 145,A 136.4166,B 20.9385,C -1.0043,E1 20.8403,E2 671.0299} C_DIS
LIN {X -96.7247,Y 79.393,Z 145,A 138.3434,B 20.9387,C -0.9994,E1 20.8369,E2 669.1062} C_DIS
LIN {X -99.5902,Y 75.7676,Z 145,A 140.4864,B 20.9389,C -0.9949,E1 20.8332,E2 666.9633} C_DIS
LIN {X -102.3072,Y 72.0561,Z 145,A 142.6025,B 20.9392,C -0.9897,E1 20.8298,E2 664.8494} C_DIS
LIN {X -104.4661,Y 68.8889,Z 145,A 144.3375,B 20.9394,C -0.9842,E1 20.8271,E2 663.1194} C_DIS
LIN {X -106.563,Y 65.5989,Z 145,A 146.1498,B 20.9396,C -0.9802,E1 20.8244,E2 661.3069} C_DIS
LIN {X -108.8774,Y 61.6822,Z 145,A 148.27,B 20.9398,C -0.9757,E1 20.8215,E2 659.186} C_DIS
LIN {X -110.7269,Y 58.2917,Z 145,A 149.8833,B 20.9403,C -0.9649,E1 20.8194,E2 657.5926} C_DIS
LIN {X -112.2157,Y 55.3714,Z 145,A 151.4871,B 20.9403,C -0.9644,E1 20.8174,E2 655.9799} C_DIS
LIN {X -114.0713,Y 51.4417,Z 145,A 153.5647,B 20.9404,C -0.9618,E1 20.8149,E2 653.8957} C_DIS
LIN {X -115.6101,Y 47.8835,Z 145,A 155.3476,B 20.9406,C -0.9568,E1 20.813,E2 652.1148} C_DIS
LIN {X -117.2648,Y 43.674,Z 145,A 157.2915,B 20.9411,C -0.9459,E1 20.8111,E2 650.1884} C_DIS
LIN {X -118.3285,Y 40.7046,Z 145,A 158.7353,B 20.9413,C -0.9415,E1 20.8097,E2 648.747} C_DIS
LIN {X -119.2905,Y 37.7926,Z 145,A 160.151,B 20.9415,C -0.9376,E1 20.8085,E2 647.3323} C_DIS
LIN {X -120.3967,Y 34.1062,Z 145,A 162.0881,B 20.9415,C -0.9387,E1 20.807,E2 645.3785} C_DIS
LIN {X -121.5667,Y 29.6662,Z 145,A 164.1968,B 20.9417,C -0.9324,E1 20.8055,E2 643.2726} C_DIS
LIN {X -122.4176,Y 25.9343,Z 145,A 165.9176,B 20.942,C -0.9257,E1 20.8045,E2 641.5582} C_DIS
LIN {X -123.157,Y 22.1545,Z 145,A 167.6235,B 20.9423,C -0.9181,E1 20.8036,E2 639.8615} C_DIS
LIN {X -123.6655,Y 19.1125,Z 145,A 169.0114,B 20.9425,C -0.9127,E1 20.803,E2 638.4786} C_DIS
LIN {X -124.0967,Y 16.0778,Z 145,A 170.4231,B 20.9427,C -0.9086,E1 20.8025,E2 637.0683} C_DIS
LIN {X -124.4545,Y 13.0265,Z 145,A 171.8345,B 20.9429,C -0.9043,E1 20.8021,E2 635.6586} C_DIS
LIN {X -124.7781,Y 9.4345,Z 145,A 173.5758,B 20.9429,C -0.9025,E1 20.8017,E2 633.9099} C_DIS
LIN {X -124.992,Y 5.9651,Z 145,A 175.237,B 20.943,C -0.9,E1 20.8014,E2 632.2434} C_DIS
LIN {X -125.1278,Y 1.4111,Z 145,A 177.2848,B 20.9434,C -0.892,E1 20.8014,E2 630.2032} C_DIS
LIN {X -125.113,Y -2.3028,Z 145,A 179.066,B 20.9434,C -0.8896,E1 20.8014,E2 628.4156} C_DIS
LIN {X -124.9724,Y -6.355,Z 145,A -179.1229,B 20.9438,C -0.8821,E1 20.8016,E2 626.6123} C_DIS
LIN {X -124.7366,Y -9.9782,Z 145,A -177.3431,B 20.9438,C -0.8812,E1 20.8019,E2 624.822} C_DIS
LIN {X -124.2857,Y -14.5469,Z 145,A -175.2915,B 20.9441,C -0.8728,E1 20.8026,E2 622.7792} C_DIS
LIN {X -123.7803,Y -18.367,Z 145,A -173.6318,B 20.9445,C -0.8634,E1 20.8032,E2 621.1338} C_DIS
LIN {X -123.2929,Y -21.395,Z 145,A -172.1984,B 20.9446,C -0.8602,E1 20.8039,E2 619.6992} C_DIS
LIN {X -122.7309,Y -24.4104,Z 145,A -170.7859,B 20.9448,C -0.8562,E1 20.8046,E2 618.2877} C_DIS
LIN {X -121.9255,Y -28.1546,Z 145,A -168.8947,B 20.9448,C -0.856,E1 20.8058,E2 616.3835} C_DIS
LIN {X -120.9232,Y -32.1871,Z 145,A -167.0305,B 20.9451,C -0.8488,E1 20.8071,E2 614.5263} C_DIS
LIN {X -119.7467,Y -36.3214,Z 145,A -164.9755,B 20.9451,C -0.8462,E1 20.8087,E2 612.4642} C_DIS
LIN {X -118.5758,Y -39.98,Z 145,A -163.3527,B 20.9456,C -0.8359,E1 20.8101,E2 610.8591} C_DIS
LIN {X -117.559,Y -42.8776,Z 145,A -161.7685,B 20.9455,C -0.8385,E1 20.8116,E2 609.2566} C_DIS
LIN {X -116.1202,Y -46.6317,Z 145,A -160.0384,B 20.9458,C -0.8291,E1 20.8134,E2 607.5413} C_DIS
LIN {X -114.708,Y -50.0059,Z 145,A -158.2421,B 20.9458,C -0.8289,E1 20.8153,E2 605.7333} C_DIS
LIN {X -113.1218,Y -53.4984,Z 145,A -156.5769,B 20.9462,C -0.8206,E1 20.8173,E2 604.0805} C_DIS
LIN {X -111.7704,Y -56.2678,Z 145,A -155.216,B 20.9464,C -0.8148,E1 20.819,E2 602.727} C_DIS
LIN {X -110.0059,Y -59.646,Z 145,A -153.2974,B 20.9464,C -0.8166,E1 20.8215,E2 600.7909} C_DIS
LIN {X -107.724,Y -63.6749,Z 145,A -151.2573,B 20.9466,C -0.808,E1 20.8243,E2 598.7621} C_DIS
LIN {X -105.721,Y -66.9474,Z 145,A -149.3864,B 20.9466,C -0.8078,E1 20.8271,E2 596.8801} C_DIS
LIN {X -103.1797,Y -70.8011,Z 145,A -147.2622,B 20.9468,C -0.8029,E1 20.8304,E2 594.7569} C_DIS
LIN {X -100.9662,Y -73.9237,Z 145,A -145.5046,B 20.947,C -0.7988,E1 20.8333,E2 593.0004} C_DIS
LIN {X -98.6656,Y -76.9681,Z 145,A -143.7328,B 20.947,C -0.7955,E1 20.8363,E2 591.2274} C_DIS
LIN {X -95.9952,Y -80.2733,Z 145,A -141.8569,B 20.9473,C -0.7884,E1 20.8396,E2 589.3612} C_DIS
LIN {X -93.4851,Y -83.1838,Z 145,A -140.0048,B 20.9473,C -0.7879,E1 20.8431,E2 587.5001} C_DIS
LIN {X -90.6283,Y -86.2868,Z 145,A -138.0773,B 20.9475,C -0.7836,E1 20.8468,E2 585.5746} C_DIS
LIN {X -87.3952,Y -89.5601,Z 145,A -136.0253,B 20.9478,C -0.7771,E1 20.8508,E2 583.5303} C_DIS
LIN {X -84.4233,Y -92.3671,Z 145,A -134.0801,B 20.9478,C -0.7762,E1 20.8548,E2 581.578} C_DIS
LIN {X -81.1513,Y -95.254,Z 145,A -132.1437,B 20.948,C -0.7699,E1 20.8589,E2 579.65} C_DIS
LIN {X -78.1829,Y -97.7056,Z 145,A -130.2968,B 20.948,C -0.7699,E1 20.8629,E2 577.7946} C_DIS
LIN {X -74.556,Y -100.5002,Z 145,A -128.1884,B 20.9481,C -0.7667,E1 20.8676,E2 575.6859} C_DIS
LIN {X -70.8344,Y -103.1569,Z 145,A -126.1235,B 20.9483,C -0.7622,E1 20.8723,E2 573.6252} C_DIS
LIN {X -67.5944,Y -105.3084,Z 145,A -124.458,B 20.9485,C -0.7549,E1 20.8762,E2 571.9737} C_DIS
LIN {X -64.3361,Y -107.3304,Z 145,A -122.5392,B 20.9484,C -0.7587,E1 20.8808,E2 570.037} C_DIS
LIN {X -60.32,Y -109.6378,Z 145,A -120.5614,B 20.9487,C -0.7501,E1 20.8855,E2 568.0762} C_DIS
LIN {X -57.6261,Y -111.0765,Z 145,A -119.1541,B 20.9487,C -0.7486,E1 20.889,E2 566.6683} C_DIS
LIN {X -54.886,Y -112.4552,Z 145,A -117.7472,B 20.9487,C -0.747,E1 20.8925,E2 565.2614} C_DIS
LIN {X -51.412,Y -114.0846,Z 145,A -115.8351,B 20.9487,C -0.7512,E1 20.8974,E2 563.3319} C_DIS
LIN {X -47.1903,Y -115.895,Z 145,A -113.8759,B 20.9489,C -0.7433,E1 20.9024,E2 561.3894} C_DIS
LIN {X -44.3207,Y -117.0225,Z 145,A -112.4697,B 20.9489,C -0.7417,E1 20.9061,E2 559.984} C_DIS
LIN {X -41.4427,Y -118.0725,Z 145,A -110.9917,B 20.9489,C -0.7435,E1 20.91,E2 558.4975} C_DIS
LIN {X -38.3643,Y -119.1078,Z 145,A -109.4474,B 20.9489,C -0.7446,E1 20.9141,E2 556.9466} C_DIS
LIN {X -34.1217,Y -120.3923,Z 145,A -107.3727,B 20.9489,C -0.745,E1 20.9197,E2 554.8668} C_DIS
LIN {X -29.6531,Y -121.5699,Z 145,A -105.2699,B 20.9489,C -0.7432,E1 20.9254,E2 552.7652} C_DIS
LIN {X -25.9181,Y -122.4211,Z 145,A -103.6686,B 20.9492,C -0.7362,E1 20.9297,E2 551.1812} C_DIS
LIN {X -22.9099,Y -123.0201,Z 145,A -102.2657,B 20.9492,C -0.7355,E1 20.9336,E2 549.7781} C_DIS
LIN {X -19.8877,Y -123.5453,Z 145,A -100.8441,B 20.9492,C -0.7358,E1 20.9375,E2 548.3543} C_DIS
LIN {X -16.8379,Y -123.9971,Z 145,A -99.4261,B 20.9492,C -0.7357,E1 20.9414,E2 546.9351} C_DIS
LIN {X -13.0312,Y -124.4539,Z 145,A -97.6926,B 20.9492,C -0.7345,E1 20.9462,E2 545.2036} C_DIS
LIN {X -9.9866,Y -124.7359,Z 145,A -96.2115,B 20.9492,C -0.7377,E1 20.9504,E2 543.7127} C_DIS
LIN {X -6.9156,Y -124.9443,Z 145,A -94.8538,B 20.9492,C -0.7356,E1 20.9541,E2 542.3604} C_DIS
LIN {X -3.0686,Y -125.097,Z 145,A -93.1271,B 20.9492,C -0.7343,E1 20.9589,E2 540.637} C_DIS
LIN {X 0.281,Y -125.1343,Z 145,A -91.465,B 20.949,C -0.7399,E1 20.9636,E2 538.9594} C_DIS
LIN {X 0.281,Y -125.1343,Z 145,A -91.465,B 20.949,C -0.7399,E1 20.9636,E2 538.9594} C_DIS
Enddeposition()
LIN {X 0.9323,Y -131.2505,Z 146,A -92.6428,B 24.9669,C -1.3301,E1 25.0017,E2 539.1317} C_DIS
Startdeposition()
$VEL.CP = VEL_PRINT
LIN {X 3.4883,Y -131.209,Z 146,A -91.2618,B 24.9662,C -1.3442,E1 25.0057,E2 537.7175} C_DIS
LIN {X 7.2765,Y -131.0552,Z 146,A -89.5355,B 24.9659,C -1.3485,E1 25.0105,E2 535.9815} C_DIS
LIN {X 11.3348,Y -130.7651,Z 146,A -87.8592,B 24.9662,C -1.3442,E1 25.0152,E2 534.3163} C_DIS
LIN {X 15.1911,Y -130.3735,Z 146,A -86.1066,B 24.9659,C -1.3484,E1 25.02,E2 532.555} C_DIS
LIN {X 19.3795,Y -129.8184,Z 146,A -84.3039,B 24.9659,C -1.3474,E1 25.025,E2 530.7561} C_DIS
LIN {X 23.0891,Y -129.2083,Z 146,A -82.6989,B 24.966,C -1.3469,E1 25.0294,E2 529.1541} C_DIS
LIN {X 26.3578,Y -128.5814,Z 146,A -81.1993,B 24.9658,C -1.3506,E1 25.0336,E2 527.6475} C_DIS
LIN {X 30.6722,Y -127.6209,Z 146,A -79.3514,B 24.966,C -1.3481,E1 25.0386,E2 525.8079} C_DIS
LIN {X 33.5348,Y -126.899,Z 146,A -78.1034,B 24.966,C -1.3473,E1 25.0419,E2 524.5637} C_DIS
LIN {X 36.7901,Y -125.9934,Z 146,A -76.4953,B 24.9656,C -1.3561,E1 25.0463,E2 522.9377} C_DIS
LIN {X 40.7318,Y -124.7772,Z 146,A -74.6508,B 24.9653,C -1.3606,E1 25.0512,E2 521.0859} C_DIS
LIN {X 44.495,Y -123.4828,Z 146,A -73.0785,B 24.9657,C -1.3541,E1 25.0553,E2 519.5321} C_DIS
LIN {X 47.1753,Y -122.4846,Z 146,A -71.7039,B 24.9652,C -1.3626,E1 25.0589,E2 518.1405} C_DIS
LIN {X 50.3693,Y -121.2056,Z 146,A -70.366,B 24.9656,C -1.356,E1 25.0624,E2 516.8212} C_DIS
LIN {X 53.4172,Y -119.8934,Z 146,A -68.8418,B 24.9652,C -1.3623,E1 25.0663,E2 515.2859} C_DIS
LIN {X 56.2649,Y -118.584,Z 146,A -67.4482,B 24.9651,C -1.3658,E1 25.0698,E2 513.8874} C_DIS
LIN {X 59.3003,Y -117.0954,Z 146,A -65.979,B 24.9649,C -1.368,E1 25.0735,E2 512.4171} C_DIS
LIN {X 62.6083,Y -115.3628,Z 146,A -64.3103,B 24.9647,C -1.3729,E1 25.0776,E2 510.7415} C_DIS
LIN {X 65.9458,Y -113.4878,Z 146,A -62.6388,B 24.9645,C -1.376,E1 25.0817,E2 509.0677} C_DIS
LIN {X 69.6531,Y -111.2514,Z 146,A -60.7489,B 24.9643,C -1.3796,E1 25.0862,E2 507.1752} C_DIS
LIN {X 73.1107,Y -109.0101,Z 146,A -58.9777,B 24.9643,C -1.3818,E1 25.0903,E2 505.4049} C_DIS
LIN {X 76.4332,Y -106.7065,Z 146,A -57.216,B 24.9641,C -1.3853,E1 25.0943,E2 503.6409} C_DIS
LIN {X 79.9343,Y -104.1098,Z 146,A -55.2829,B 24.9638,C -1.3911,E1 25.0987,E2 501.7012} C_DIS
LIN {X 83.3978,Y -101.3571,Z 146,A -53.3745,B 24.9636,C -1.3942,E1 25.1028,E2 499.7926} C_DIS
LIN {X 86.4108,Y -98.8003,Z 146,A -51.7093,B 24.9636,C -1.395,E1 25.1063,E2 498.132} C_DIS
LIN {X 89.4925,Y -96.0177,Z 146,A -49.9122,B 24.9634,C -1.3985,E1 25.11,E2 496.3339} C_DIS
LIN {X 92.2691,Y -93.3532,Z 146,A -48.1579,B 24.9629,C -1.4067,E1 25.1135,E2 494.5676} C_DIS
LIN {X 95.2921,Y -90.265,Z 146,A -46.3327,B 24.9629,C -1.4081,E1 25.1171,E2 492.7468} C_DIS
LIN {X 98.1378,Y -87.1628,Z 146,A -44.4719,B 24.9625,C -1.4142,E1 25.1206,E2 490.8801} C_DIS
LIN {X 101.0444,Y -83.7755,Z 146,A -42.6031,B 24.9625,C -1.4151,E1 25.1239,E2 489.0178} C_DIS
LIN {X 103.4663,Y -80.7662,Z 146,A -40.926,B 24.9623,C -1.4192,E1 25.1268,E2 487.3389} C_DIS
LIN {X 106.0029,Y -77.4068,Z 146,A -39.0522,B 24.9619,C -1.4263,E1 25.13,E2 485.4573} C_DIS
LIN {X 108.487,Y -73.8851,Z 146,A -37.199,B 24.9617,C -1.4301,E1 25.1329,E2 483.6043} C_DIS
LIN {X 110.8548,Y -70.2821,Z 146,A -35.2752,B 24.9613,C -1.4378,E1 25.1358,E2 481.6718} C_DIS
LIN {X 113.095,Y -66.6172,Z 146,A -33.4795,B 24.9613,C -1.439,E1 25.1384,E2 479.8825} C_DIS
LIN {X 114.9392,Y -63.3824,Z 146,A -31.8788,B 24.961,C -1.4425,E1 25.1406,E2 478.2819} C_DIS
LIN {X 116.7345,Y -60.0093,Z 146,A -30.1824,B 24.9607,C -1.4492,E1 25.1428,E2 476.5788} C_DIS
LIN {X 118.3456,Y -56.764,Z 146,A -28.7625,B 24.9609,C -1.4451,E1 25.1445,E2 475.1759} C_DIS
LIN {X 119.7853,Y -53.6589,Z 146,A -27.2601,B 24.9606,C -1.4502,E1 25.1463,E2 473.6697} C_DIS
LIN {X 120.9151,Y -51.0648,Z 146,A -25.8877,B 24.96,C -1.4616,E1 25.1478,E2 472.278} C_DIS
LIN {X 122.1991,Y -47.9098,Z 146,A -24.5229,B 24.96,C -1.4596,E1 25.1492,E2 470.9255} C_DIS
LIN {X 123.3999,Y -44.7252,Z 146,A -23.0992,B 24.96,C -1.4609,E1 25.1506,E2 469.5067} C_DIS
LIN {X 124.5178,Y -41.5108,Z 146,A -21.5676,B 24.9596,C -1.4682,E1 25.1519,E2 467.9666} C_DIS
LIN {X 125.4868,Y -38.4827,Z 146,A -20.2045,B 24.9594,C -1.4713,E1 25.1531,E2 466.6039} C_DIS
LIN {X 126.3487,Y -35.5512,Z 146,A -18.8087,B 24.959,C -1.479,E1 25.1542,E2 465.1978} C_DIS
LIN {X 127.3107,Y -31.9371,Z 146,A -17.2395,B 24.959,C -1.4808,E1 25.1553,E2 463.6334} C_DIS
LIN {X 128.4679,Y -26.9153,Z 146,A -14.7178,B 24.9577,C -1.5032,E1 25.1568,E2 461.0737} C_DIS
LIN {X 129.4334,Y -21.7924,Z 146,A -12.6958,B 24.958,C -1.4967,E1 25.1578,E2 459.0788} C_DIS
LIN {X 130.0108,Y -18.0379,Z 146,A -11.0614,B 24.9578,C -1.5008,E1 25.1584,E2 457.4443} C_DIS
LIN {X 130.4849,Y -14.1989,Z 146,A -9.4786,B 24.9578,C -1.5006,E1 25.1589,E2 455.8714} C_DIS
LIN {X 130.7694,Y -11.2844,Z 146,A -8.0591,B 24.9571,C -1.5126,E1 25.1593,E2 454.4321} C_DIS
LIN {X 131.0613,Y -7.1533,Z 146,A -6.2846,B 24.9569,C -1.5167,E1 25.1596,E2 452.6583} C_DIS
LIN {X 131.2013,Y -3.7635,Z 146,A -4.8506,B 24.9568,C -1.5191,E1 25.1597,E2 451.2274} C_DIS
LIN {X 131.259,Y 0.1911,Z 146,A -2.963,B 24.9559,C -1.5336,E1 25.1597,E2 449.3168} C_DIS
LIN {X 131.1744,Y 4.6306,Z 146,A -1.1811,B 24.9561,C -1.5314,E1 25.1597,E2 447.5506} C_DIS
LIN {X 131.0108,Y 8.006,Z 146,A 0.2363,B 24.956,C -1.5331,E1 25.1594,E2 446.1377} C_DIS
LIN {X 130.7095,Y 11.9696,Z 146,A 2.0147,B 24.9555,C -1.5411,E1 25.159,E2 444.3508} C_DIS
LIN {X 130.2392,Y 16.3157,Z 146,A 3.8168,B 24.9555,C -1.5415,E1 25.1584,E2 442.5586} C_DIS
LIN {X 129.8562,Y 19.1196,Z 146,A 5.0475,B 24.9553,C -1.5453,E1 25.1579,E2 441.3262} C_DIS
LIN {X 129.0311,Y 24.0664,Z 146,A 7.46,B 24.9541,C -1.5646,E1 25.1568,E2 438.8823} C_DIS
LIN {X 128.0309,Y 28.9145,Z 146,A 9.3553,B 24.9546,C -1.5569,E1 25.1557,E2 437.0163} C_DIS
LIN {X 127.3086,Y 31.9454,Z 146,A 10.7938,B 24.9541,C -1.5655,E1 25.1547,E2 435.5658} C_DIS
LIN {X 126.4297,Y 35.2618,Z 146,A 12.1836,B 24.9541,C -1.5643,E1 25.1537,E2 434.1868} C_DIS
LIN {X 125.6094,Y 38.082,Z 146,A 13.4758,B 24.9539,C -1.5688,E1 25.1527,E2 432.8914} C_DIS
LIN {X 124.5383,Y 41.4494,Z 146,A 14.9882,B 24.9537,C -1.5719,E1 25.1514,E2 431.3802} C_DIS
LIN {X 123.6128,Y 44.1347,Z 146,A 16.3543,B 24.9531,C -1.5826,E1 25.1501,E2 429.9966} C_DIS
LIN {X 122.5643,Y 46.9703,Z 146,A 17.7364,B 24.9526,C -1.5899,E1 25.1487,E2 428.6049} C_DIS
LIN {X 120.7621,Y 51.428,Z 146,A 19.7787,B 24.9524,C -1.593,E1 25.1465,E2 426.5664} C_DIS
LIN {X 119.1334,Y 55.091,Z 146,A 21.3897,B 24.9526,C -1.5906,E1 25.1447,E2 424.9699} C_DIS
LIN {X 117.7713,Y 57.946,Z 146,A 22.8069,B 24.9522,C -1.5966,E1 25.1429,E2 423.5463} C_DIS
LIN {X 116.207,Y 61.0223,Z 146,A 24.2606,B 24.9522,C -1.598,E1 25.1411,E2 422.097} C_DIS
LIN {X 114.3071,Y 64.5155,Z 146,A 26.0895,B 24.9516,C -1.6078,E1 25.1386,E2 420.2544} C_DIS
LIN {X 112.0872,Y 68.3002,Z 146,A 28.0513,B 24.9511,C -1.6156,E1 25.1358,E2 418.2844} C_DIS
LIN {X 109.6617,Y 72.1291,Z 146,A 29.9332,B 24.9511,C -1.6156,E1 25.1329,E2 416.4118} C_DIS
LIN {X 107.4213,Y 75.4257,Z 146,A 31.7377,B 24.9506,C -1.6236,E1 25.13,E2 414.5972} C_DIS
LIN {X 104.9067,Y 78.8856,Z 146,A 33.5723,B 24.9504,C -1.6266,E1 25.127,E2 412.7644} C_DIS
LIN {X 102.474,Y 82.0213,Z 146,A 35.2468,B 24.9504,C -1.6277,E1 25.1241,E2 411.0952} C_DIS
LIN {X 99.8794,Y 85.1612,Z 146,A 37.0147,B 24.9501,C -1.6314,E1 25.1209,E2 409.3266} C_DIS
LIN {X 97.1248,Y 88.2897,Z 146,A 38.8156,B 24.9499,C -1.6347,E1 25.1176,E2 407.5261} C_DIS
LIN {X 94.5031,Y 91.0908,Z 146,A 40.5538,B 24.9495,C -1.6418,E1 25.1142,E2 405.7785} C_DIS
LIN {X 91.5432,Y 94.0652,Z 146,A 42.3742,B 24.9493,C -1.6452,E1 25.1106,E2 403.9578} C_DIS
LIN {X 88.6205,Y 96.8234,Z 146,A 44.0791,B 24.9493,C -1.6463,E1 25.1071,E2 402.2573} C_DIS
LIN {X 85.3967,Y 99.6785,Z 146,A 46.0163,B 24.9488,C -1.6531,E1 25.103,E2 400.3117} C_DIS
LIN {X 82.2543,Y 102.2867,Z 146,A 47.734,B 24.9488,C -1.6531,E1 25.0993,E2 398.6005} C_DIS
LIN {X 79.0104,Y 104.8125,Z 146,A 49.4718,B 24.9488,C -1.6534,E1 25.0955,E2 396.8683} C_DIS
LIN {X 75.8931,Y 107.0917,Z 146,A 51.2528,B 24.9483,C -1.6614,E1 25.0914,E2 395.0747} C_DIS
LIN {X 72.2132,Y 109.6064,Z 146,A 53.1242,B 24.9483,C -1.6607,E1 25.0871,E2 393.2112} C_DIS
LIN {X 68.7868,Y 111.7887,Z 146,A 54.8584,B 24.9483,C -1.6615,E1 25.083,E2 391.4808} C_DIS
LIN {X 65.2417,Y 113.8941,Z 146,A 56.7236,B 24.9479,C -1.6676,E1 25.0785,E2 389.6067} C_DIS
LIN {X 62.7693,Y 115.275,Z 146,A 58.4158,B 24.9463,C -1.6934,E1 25.0742,E2 387.8582} C_DIS
LIN {X 58.7257,Y 117.3866,Z 146,A 60.3856,B 24.9462,C -1.6949,E1 25.0693,E2 385.8904} C_DIS
LIN {X 54.777,Y 119.2786,Z 146,A 61.7805,B 24.9477,C -1.67,E1 25.0659,E2 384.5579} C_DIS
LIN {X 51.2216,Y 120.8496,Z 146,A 63.5454,B 24.9474,C -1.6754,E1 25.0613,E2 382.7844} C_DIS
LIN {X 48.0256,Y 122.154,Z 146,A 65.0099,B 24.9474,C -1.6748,E1 25.0576,E2 381.3246} C_DIS
LIN {X 44.8414,Y 123.358,Z 146,A 66.4493,B 24.9474,C -1.6738,E1 25.0538,E2 379.8906} C_DIS
LIN {X 41.6122,Y 124.484,Z 146,A 67.8606,B 24.9477,C -1.6709,E1 25.0501,E2 378.489} C_DIS
LIN {X 38.8004,Y 125.3895,Z 146,A 69.289,B 24.9472,C -1.6791,E1 25.0462,E2 377.0437} C_DIS
LIN {X 35.352,Y 126.4044,Z 146,A 70.885,B 24.947,C -1.6816,E1 25.0419,E2 375.4444} C_DIS
LIN {X 30.9493,Y 127.5541,Z 146,A 72.8099,B 24.9471,C -1.6797,E1 25.0368,E2 373.5271} C_DIS
LIN {X 27.1453,Y 128.4185,Z 146,A 74.5067,B 24.9471,C -1.6802,E1 25.0321,E2 371.8312} C_DIS
LIN {X 23.425,Y 129.1481,Z 146,A 76.0467,B 24.9474,C -1.675,E1 25.0279,E2 370.3053} C_DIS
LIN {X 20.0798,Y 129.71,Z 146,A 77.6271,B 24.9471,C -1.6806,E1 25.0236,E2 368.7131} C_DIS
LIN {X 15.8744,Y 130.292,Z 146,A 79.4843,B 24.9471,C -1.6812,E1 25.0184,E2 366.856} C_DIS
LIN {X 11.9804,Y 130.7085,Z 146,A 81.2515,B 24.9468,C -1.6844,E1 25.0135,E2 365.0824} C_DIS
LIN {X 8.1293,Y 131.0032,Z 146,A 82.8874,B 24.947,C -1.6819,E1 25.0089,E2 363.4532} C_DIS
LIN {X 3.9565,Y 131.196,Z 146,A 84.738,B 24.947,C -1.6832,E1 25.0038,E2 361.6001} C_DIS
LIN {X -0.2205,Y 131.2561,Z 146,A 86.5901,B 24.9468,C -1.6843,E1 24.9986,E2 359.7455} C_DIS
LIN {X -4.5069,Y 131.1792,Z 146,A 88.4568,B 24.9468,C -1.6835,E1 24.9934,E2 357.8805} C_DIS
LIN {X -8.4609,Y 130.9828,Z 146,A 90.2124,B 24.9468,C -1.6842,E1 24.9885,E2 356.1225} C_DIS
LIN {X -12.5464,Y 130.6541,Z 146,A 91.9167,B 24.9472,C -1.6791,E1 24.9838,E2 354.4296} C_DIS
LIN {X -16.8199,Y 130.1731,Z 146,A 93.6924,B 24.9476,C -1.6729,E1 24.9789,E2 352.6675} C_DIS
LIN {X -20.1293,Y 129.7024,Z 146,A 95.2761,B 24.9472,C -1.6781,E1 24.9745,E2 351.0699} C_DIS
LIN {X -24.3273,Y 128.9812,Z 146,A 97.1091,B 24.9474,C -1.6754,E1 24.9695,E2 349.2416} C_DIS
LIN {X -27.8426,Y 128.268,Z 146,A 98.6862,B 24.9474,C -1.6746,E1 24.9651,E2 347.6645} C_DIS
LIN {X -31.587,Y 127.3995,Z 146,A 100.4444,B 24.9474,C -1.677,E1 24.9604,E2 345.8983} C_DIS
LIN {X -34.9359,Y 126.5208,Z 146,A 101.9322,B 24.9474,C -1.6742,E1 24.9564,E2 344.4147} C_DIS
LIN {X -38.343,Y 125.5295,Z 146,A 103.3471,B 24.948,C -1.6658,E1 24.9526,E2 343.0174} C_DIS
LIN {X -40.9031,Y 124.7202,Z 146,A 104.6686,B 24.9476,C -1.6718,E1 24.9491,E2 341.6793} C_DIS
LIN {X -44.107,Y 123.6228,Z 146,A 106.1306,B 24.9478,C -1.6691,E1 24.9452,E2 340.2208} C_DIS
LIN {X -47.2718,Y 122.4471,Z 146,A 107.5894,B 24.948,C -1.6664,E1 24.9414,E2 338.7654} C_DIS
LIN {X -50.3752,Y 121.2031,Z 146,A 108.9186,B 24.9485,C -1.6578,E1 24.938,E2 337.4535} C_DIS
LIN {X -53.4178,Y 119.8932,Z 146,A 110.4677,B 24.9483,C -1.6608,E1 24.934,E2 335.8939} C_DIS
LIN {X -56.3259,Y 118.5549,Z 146,A 111.7842,B 24.9487,C -1.6546,E1 24.9307,E2 334.5887} C_DIS
LIN {X -59.9444,Y 116.7675,Z 146,A 113.7485,B 24.9483,C -1.6616,E1 24.9258,E2 332.6024} C_DIS
LIN {X -64.2325,Y 114.4661,Z 146,A 115.7853,B 24.9488,C -1.6536,E1 24.9208,E2 330.5789} C_DIS
LIN {X -67.5699,Y 112.529,Z 146,A 117.5627,B 24.9487,C -1.655,E1 24.9165,E2 328.7928} C_DIS
LIN {X -71.2745,Y 110.2193,Z 146,A 119.4264,B 24.949,C -1.6493,E1 24.9122,E2 326.9368} C_DIS
LIN {X -74.4207,Y 108.1198,Z 146,A 121.0695,B 24.9493,C -1.6455,E1 24.9084,E2 325.297} C_DIS
LIN {X -77.9554,Y 105.5999,Z 146,A 123.0139,B 24.9493,C -1.644,E1 24.904,E2 323.3495} C_DIS
LIN {X -81.3898,Y 102.9765,Z 146,A 124.9487,B 24.9495,C -1.6422,E1 24.8997,E2 321.4117} C_DIS
LIN {X -84.6373,Y 100.3242,Z 146,A 126.7241,B 24.9499,C -1.6354,E1 24.8959,E2 319.6458} C_DIS
LIN {X -87.8862,Y 97.491,Z 146,A 128.647,B 24.95,C -1.633,E1 24.8919,E2 317.721} C_DIS
LIN {X -90.7276,Y 94.8514,Z 146,A 130.3208,B 24.9503,C -1.628,E1 24.8885,E2 316.0522} C_DIS
LIN {X -93.6914,Y 91.925,Z 146,A 132.1294,B 24.9506,C -1.6231,E1 24.8849,E2 314.2477} C_DIS
LIN {X -96.4365,Y 89.0414,Z 146,A 133.9526,B 24.9506,C -1.6228,E1 24.8814,E2 312.4172} C_DIS
LIN {X -99.2207,Y 85.9283,Z 146,A 135.7953,B 24.9509,C -1.619,E1 24.8781,E2 310.5753} C_DIS
LIN {X -102.153,Y 82.42,Z 146,A 137.6797,B 24.9515,C -1.6083,E1 24.8747,E2 308.7077} C_DIS
LIN {X -104.6636,Y 79.2076,Z 146,A 139.5629,B 24.9515,C -1.6083,E1 24.8715,E2 306.8152} C_DIS
LIN {X -107.3735,Y 75.4934,Z 146,A 141.5066,B 24.952,C -1.5997,E1 24.8684,E2 304.8827} C_DIS
LIN {X -109.7722,Y 71.9614,Z 146,A 143.3736,B 24.9524,C -1.5946,E1 24.8655,E2 303.0187} C_DIS
LIN {X -112.0348,Y 68.3855,Z 146,A 145.3141,B 24.9524,C -1.5937,E1 24.8626,E2 301.0704} C_DIS
LIN {X -114.2027,Y 64.7007,Z 146,A 147.1226,B 24.9529,C -1.5854,E1 24.8601,E2 299.2722} C_DIS
LIN {X -116.0484,Y 61.3244,Z 146,A 148.6977,B 24.9535,C -1.5754,E1 24.858,E2 297.7126} C_DIS
LIN {X -117.6206,Y 58.2514,Z 146,A 150.0422,B 24.9542,C -1.5631,E1 24.8564,E2 296.3902} C_DIS
LIN {X -118.7881,Y 55.8378,Z 146,A 151.601,B 24.9533,C -1.578,E1 24.8544,E2 294.7873} C_DIS
LIN {X -120.3898,Y 52.2891,Z 146,A 153.1323,B 24.9541,C -1.5647,E1 24.8527,E2 293.2793} C_DIS
LIN {X -121.5776,Y 49.466,Z 146,A 154.5055,B 24.9543,C -1.5623,E1 24.8513,E2 291.9043} C_DIS
LIN {X -122.8255,Y 46.2793,Z 146,A 156.0744,B 24.9543,C -1.5612,E1 24.8497,E2 290.3293} C_DIS
LIN {X -123.9365,Y 43.2161,Z 146,A 157.4379,B 24.9548,C -1.5538,E1 24.8484,E2 288.9754} C_DIS
LIN {X -124.9999,Y 40.0359,Z 146,A 158.9463,B 24.9549,C -1.5513,E1 24.8471,E2 287.4645} C_DIS
LIN {X -125.9344,Y 36.9916,Z 146,A 160.2676,B 24.9554,C -1.5435,E1 24.8461,E2 286.1541} C_DIS
LIN {X -126.7054,Y 34.2608,Z 146,A 161.6588,B 24.9552,C -1.5468,E1 24.845,E2 284.747} C_DIS
LIN {X -127.5493,Y 30.969,Z 146,A 163.0022,B 24.9558,C -1.5353,E1 24.8441,E2 283.4231} C_DIS
LIN {X -128.2683,Y 27.8413,Z 146,A 164.5163,B 24.9558,C -1.5361,E1 24.8432,E2 281.8981} C_DIS
LIN {X -129.0298,Y 24.0731,Z 146,A 166.2542,B 24.9559,C -1.5335,E1 24.8423,E2 280.1563} C_DIS
LIN {X -129.6862,Y 20.234,Z 146,A 167.8214,B 24.9566,C -1.5216,E1 24.8416,E2 278.6082} C_DIS
LIN {X -130.1164,Y 17.2529,Z 146,A 169.2442,B 24.9566,C -1.5224,E1 24.841,E2 277.1749} C_DIS
LIN {X -130.5681,Y 13.4263,Z 146,A 171.0334,B 24.9566,C -1.5219,E1 24.8405,E2 275.3761} C_DIS
LIN {X -130.9623,Y 8.7932,Z 146,A 173.0402,B 24.957,C -1.5141,E1 24.8401,E2 273.3758} C_DIS
LIN {X -131.1202,Y 5.9829,Z 146,A 174.1378,B 24.9576,C -1.5038,E1 24.8399,E2 272.2962} C_DIS
LIN {X -131.2306,Y 2.5731,Z 146,A 175.8381,B 24.9573,C -1.509,E1 24.8398,E2 270.5733} C_DIS
LIN {X -131.2325,Y -2.4599,Z 146,A 177.949,B 24.958,C -1.4976,E1 24.8398,E2 268.4767} C_DIS
LIN {X -131.1015,Y -6.354,Z 146,A 179.6078,B 24.9584,C -1.4901,E1 24.84,E2 266.8261} C_DIS
LIN {X -130.8934,Y -9.7397,Z 146,A -178.8579,B 24.9585,C -1.4878,E1 24.8403,E2 265.288} C_DIS
LIN {X -130.53,Y -13.7802,Z 146,A -177.1181,B 24.9589,C -1.4805,E1 24.8408,E2 263.555} C_DIS
LIN {X -130.1217,Y -17.2121,Z 146,A -175.5625,B 24.9591,C -1.4779,E1 24.8413,E2 261.9964} C_DIS
LIN {X -129.528,Y -21.2257,Z 146,A -173.7643,B 24.9593,C -1.4735,E1 24.8421,E2 260.1981} C_DIS
LIN {X -128.8963,Y -24.7715,Z 146,A -172.1804,B 24.9596,C -1.469,E1 24.8429,E2 258.6154} C_DIS
LIN {X -128.0233,Y -28.9478,Z 146,A -170.408,B 24.9601,C -1.4588,E1 24.844,E2 256.857} C_DIS
LIN {X -127.215,Y -32.314,Z 146,A -168.7854,B 24.9601,C -1.4593,E1 24.845,E2 255.2235} C_DIS
LIN {X -126.1947,Y -36.1018,Z 146,A -166.9353,B 24.9601,C -1.4606,E1 24.8464,E2 253.3596} C_DIS
LIN {X -125.136,Y -39.6099,Z 146,A -165.4315,B 24.9606,C -1.4511,E1 24.8477,E2 251.8699} C_DIS
LIN {X -124.0936,Y -42.7629,Z 146,A -164.1285,B 24.9612,C -1.4396,E1 24.8488,E2 250.5868} C_DIS
LIN {X -122.9785,Y -45.8708,Z 146,A -162.5907,B 24.9612,C -1.4399,E1 24.8503,E2 249.0396} C_DIS
LIN {X -121.87,Y -48.7406,Z 146,A -161.171,B 24.9612,C -1.4396,E1 24.8518,E2 247.6127} C_DIS
LIN {X -120.5377,Y -51.9469,Z 146,A -159.7132,B 24.9616,C -1.4323,E1 24.8534,E2 246.1641} C_DIS
LIN {X -119.2522,Y -54.8341,Z 146,A -158.3007,B 24.9616,C -1.4299,E1 24.855,E2 244.7497} C_DIS
LIN {X -117.7779,Y -57.9325,Z 146,A -156.7843,B 24.9619,C -1.4265,E1 24.8568,E2 243.2332} C_DIS
LIN {X -116.2141,Y -61.0088,Z 146,A -155.3877,B 24.9624,C -1.4169,E1 24.8586,E2 241.8519} C_DIS
LIN {X -114.3548,Y -64.4305,Z 146,A -153.5701,B 24.9624,C -1.4179,E1 24.8611,E2 240.0225} C_DIS
LIN {X -112.3526,Y -67.8617,Z 146,A -151.7837,B 24.9624,C -1.4157,E1 24.8636,E2 238.2321} C_DIS
LIN {X -110.2452,Y -71.2347,Z 146,A -150.0247,B 24.9626,C -1.4122,E1 24.8663,E2 236.4725} C_DIS
LIN {X -107.9991,Y -74.5966,Z 146,A -148.2945,B 24.963,C -1.4059,E1 24.869,E2 234.7487} C_DIS
LIN {X -105.5714,Y -77.9942,Z 146,A -146.4084,B 24.963,C -1.4044,E1 24.8721,E2 232.857} C_DIS
LIN {X -103.2047,Y -81.0993,Z 146,A -144.6987,B 24.9633,C -1.4004,E1 24.875,E2 231.1486} C_DIS
LIN {X -100.345,Y -84.6125,Z 146,A -142.6783,B 24.9634,C -1.3978,E1 24.8786,E2 229.1252} C_DIS
LIN {X -97.7157,Y -87.6353,Z 146,A -140.9564,B 24.9637,C -1.3924,E1 24.8818,E2 227.4083} C_DIS
LIN {X -94.7772,Y -90.8053,Z 146,A -139.1063,B 24.964,C -1.3864,E1 24.8853,E2 225.5646} C_DIS
LIN {X -91.8129,Y -93.8014,Z 146,A -137.2527,B 24.9642,C -1.383,E1 24.889,E2 223.711} C_DIS
LIN {X -88.9468,Y -96.5235,Z 146,A -135.6188,B 24.9646,C -1.3749,E1 24.8923,E2 222.0898} C_DIS
LIN {X -86.1442,Y -99.0329,Z 146,A -133.8063,B 24.9643,C -1.38,E1 24.8961,E2 220.2579} C_DIS
LIN {X -83.0135,Y -101.6713,Z 146,A -132.0598,B 24.9646,C -1.3746,E1 24.8999,E2 218.5177} C_DIS
LIN {X -79.8422,Y -104.1803,Z 146,A -130.3136,B 24.9648,C -1.3704,E1 24.9037,E2 216.7752} C_DIS
LIN {X -76.7705,Y -106.4645,Z 146,A -128.5492,B 24.9648,C -1.3721,E1 24.9077,E2 215.0004} C_DIS
LIN {X -73.4378,Y -108.7897,Z 146,A -126.8156,B 24.965,C -1.3671,E1 24.9117,E2 213.2729} C_DIS
LIN {X -69.731,Y -111.2027,Z 146,A -124.8455,B 24.965,C -1.366,E1 24.9163,E2 211.2991} C_DIS
LIN {X -66.3443,Y -113.2553,Z 146,A -123.1526,B 24.9653,C -1.3616,E1 24.9204,E2 209.6114} C_DIS
LIN {X -62.5229,Y -115.4094,Z 146,A -121.164,B 24.9653,C -1.3627,E1 24.9252,E2 207.6147} C_DIS
LIN {X -59.0003,Y -117.2481,Z 146,A -119.4227,B 24.9653,C -1.3608,E1 24.9296,E2 205.8732} C_DIS
LIN {X -55.2152,Y -119.076,Z 146,A -117.7534,B 24.9659,C -1.3502,E1 24.9337,E2 204.2246} C_DIS
LIN {X -52.1938,Y -120.431,Z 146,A -116.2784,B 24.9659,C -1.3501,E1 24.9375,E2 202.7464} C_DIS
LIN {X -49.4115,Y -121.5996,Z 146,A -115.0181,B 24.9661,C -1.3458,E1 24.9407,E2 201.4934} C_DIS
LIN {X -46.2619,Y -122.8321,Z 146,A -113.5234,B 24.9661,C -1.3453,E1 24.9447,E2 199.9968} C_DIS
LIN {X -43.0051,Y -124.0096,Z 146,A -111.9797,B 24.9661,C -1.3456,E1 24.9487,E2 198.4493} C_DIS
LIN {X -39.9669,Y -125.0219,Z 146,A -110.641,B 24.9663,C -1.3415,E1 24.9523,E2 197.118} C_DIS
LIN {X -36.8143,Y -125.9863,Z 146,A -109.0686,B 24.966,C -1.3472,E1 24.9565,E2 195.5293} C_DIS
LIN {X -32.7008,Y -127.1168,Z 146,A -107.2066,B 24.966,C -1.346,E1 24.9615,E2 193.6674} C_DIS
LIN {X -29.461,Y -127.9061,Z 146,A -105.7832,B 24.9662,C -1.3436,E1 24.9654,E2 192.2478} C_DIS
LIN {X -26.3763,Y -128.5776,Z 146,A -104.3728,B 24.9662,C -1.3446,E1 24.9693,E2 190.8332} C_DIS
LIN {X -22.6407,Y -129.2885,Z 146,A -102.6019,B 24.9659,C -1.3497,E1 24.9742,E2 189.0483} C_DIS
LIN {X -18.9142,Y -129.8856,Z 146,A -101.1701,B 24.9665,C -1.3382,E1 24.978,E2 187.6427} C_DIS
LIN {X -15.5677,Y -130.3286,Z 146,A -99.6437,B 24.9663,C -1.3406,E1 24.9823,E2 186.1094} C_DIS
LIN {X -12.0142,Y -130.7052,Z 146,A -97.9299,B 24.9659,C -1.3484,E1 24.9871,E2 184.3761} C_DIS
LIN {X -7.5655,Y -131.0379,Z 146,A -96.0669,B 24.9662,C -1.3441,E1 24.9923,E2 182.5229} C_DIS
LIN {X -3.6647,Y -131.2041,Z 146,A -94.3736,B 24.9662,C -1.3437,E1 24.997,E2 180.8301} C_DIS
LIN {X 0.4486,Y -131.2548,Z 146,A -92.6653,B 24.9664,C -1.3396,E1 25.0017,E2 179.1317} C_DIS
LIN {X 0.4486,Y -131.2548,Z 146,A -92.6653,B 24.9664,C -1.3396,E1 25.0017,E2 179.1317} C_DIS
Enddeposition()
LIN {X 0.9217,Y -130.2941,Z 146,A -92.5622,B 24.9658,C -1.351,E1 25.0021,E2 179.0016} C_DIS
Startdeposition()
$VEL.CP = VEL_PRINT
LIN {X -2.1677,Y -130.2803,Z 146,A -94.4731,B 24.9672,C -1.3224,E1 24.9966,E2 180.9802} C_DIS
LIN {X -5.5174,Y -130.1822,Z 146,A -96.0235,B 24.9674,C -1.3183,E1 24.9922,E2 182.5405} C_DIS
LIN {X -9.421,Y -129.9572,Z 146,A -97.6233,B 24.9672,C -1.3243,E1 24.9878,E2 184.1266} C_DIS
LIN {X -12.7467,Y -129.6736,Z 146,A -99.1215,B 24.9672,C -1.3229,E1 24.9836,E2 185.629} C_DIS
LIN {X -16.7188,Y -129.2213,Z 146,A -100.8898,B 24.9672,C -1.3227,E1 24.9787,E2 187.399} C_DIS
LIN {X -20.0238,Y -128.7504,Z 146,A -102.356,B 24.9672,C -1.3231,E1 24.9747,E2 188.8654} C_DIS
LIN {X -23.7098,Y -128.125,Z 146,A -103.9609,B 24.9671,C -1.3256,E1 24.9703,E2 190.466} C_DIS
LIN {X -26.7389,Y -127.5273,Z 146,A -105.322,B 24.9671,C -1.326,E1 24.9665,E2 191.8277} C_DIS
LIN {X -29.7743,Y -126.8529,Z 146,A -106.6928,B 24.9671,C -1.3265,E1 24.9628,E2 193.199} C_DIS
LIN {X -32.8133,Y -126.101,Z 146,A -108.0732,B 24.9671,C -1.3272,E1 24.9591,E2 194.5799} C_DIS
LIN {X -35.8532,Y -125.2706,Z 146,A -109.4628,B 24.967,C -1.3279,E1 24.9553,E2 195.97} C_DIS
LIN {X -38.3458,Y -124.5279,Z 146,A -110.6063,B 24.967,C -1.3288,E1 24.9523,E2 197.1133} C_DIS
LIN {X -41.5656,Y -123.491,Z 146,A -112.0822,B 24.9668,C -1.3305,E1 24.9484,E2 198.5877} C_DIS
LIN {X -44.6528,Y -122.4087,Z 146,A -113.5215,B 24.9668,C -1.3318,E1 24.9446,E2 200.0269} C_DIS
LIN {X -47.5119,Y -121.327,Z 146,A -114.9063,B 24.9668,C -1.3311,E1 24.9409,E2 201.4163} C_DIS
LIN {X -50.5646,Y -120.087,Z 146,A -116.3731,B 24.9668,C -1.3317,E1 24.9372,E2 202.885} C_DIS
LIN {X -53.6645,Y -118.7346,Z 146,A -117.8565,B 24.9667,C -1.3336,E1 24.9334,E2 204.3675} C_DIS
LIN {X -56.4154,Y -117.4516,Z 146,A -119.1972,B 24.9667,C -1.3349,E1 24.93,E2 205.7085} C_DIS
LIN {X -59.579,Y -115.8797,Z 146,A -120.7445,B 24.9665,C -1.3372,E1 24.9261,E2 207.2545} C_DIS
LIN {X -62.7582,Y -114.191,Z 146,A -122.469,B 24.9668,C -1.3324,E1 24.9219,E2 208.9953} C_DIS
LIN {X -66.6068,Y -111.9891,Z 146,A -124.3641,B 24.9665,C -1.3379,E1 24.9173,E2 210.8829} C_DIS
LIN {X -70.1145,Y -109.8271,Z 146,A -126.2046,B 24.9665,C -1.3393,E1 24.9129,E2 212.7259} C_DIS
LIN {X -73.73,Y -107.4332,Z 146,A -128.0794,B 24.9662,C -1.344,E1 24.9086,E2 214.5957} C_DIS
LIN {X -77.1437,Y -105.0089,Z 146,A -129.9329,B 24.966,C -1.3466,E1 24.9044,E2 216.4495} C_DIS
LIN {X -80.4855,Y -102.4699,Z 146,A -131.7866,B 24.9659,C -1.3496,E1 24.9003,E2 218.3028} C_DIS
LIN {X -83.6035,Y -99.9425,Z 146,A -133.6014,B 24.9659,C -1.3506,E1 24.8964,E2 220.1223} C_DIS
LIN {X -86.9316,Y -97.0613,Z 146,A -135.5036,B 24.9656,C -1.3561,E1 24.8924,E2 222.0189} C_DIS
LIN {X -90.1053,Y -94.1225,Z 146,A -137.4365,B 24.9654,C -1.3586,E1 24.8885,E2 223.9537} C_DIS
LIN {X -93.2814,Y -90.9765,Z 146,A -139.4293,B 24.9653,C -1.3616,E1 24.8846,E2 225.9479} C_DIS
LIN {X -96.2138,Y -87.8697,Z 146,A -141.31,B 24.9651,C -1.3657,E1 24.881,E2 227.827} C_DIS
LIN {X -99.0038,Y -84.7138,Z 146,A -143.1712,B 24.9649,C -1.3696,E1 24.8776,E2 229.6873} C_DIS
LIN {X -101.687,Y -81.4735,Z 146,A -145.0298,B 24.9647,C -1.3737,E1 24.8743,E2 231.5449} C_DIS
LIN {X -104.2597,Y -78.1542,Z 146,A -146.9232,B 24.9645,C -1.376,E1 24.8711,E2 233.4418} C_DIS
LIN {X -106.8762,Y -74.5352,Z 146,A -148.8355,B 24.9641,C -1.3835,E1 24.868,E2 235.3455} C_DIS
LIN {X -109.2327,Y -71.0368,Z 146,A -150.7075,B 24.9639,C -1.3876,E1 24.8651,E2 237.2173} C_DIS
LIN {X -111.5821,Y -67.2864,Z 146,A -152.6757,B 24.9637,C -1.3918,E1 24.8622,E2 239.1856} C_DIS
LIN {X -113.7905,Y -63.4816,Z 146,A -154.6219,B 24.9635,C -1.3965,E1 24.8596,E2 241.1306} C_DIS
LIN {X -115.6881,Y -59.9521,Z 146,A -156.2948,B 24.963,C -1.4057,E1 24.8574,E2 242.7905} C_DIS
LIN {X -117.085,Y -57.1742,Z 146,A -157.6698,B 24.9628,C -1.4093,E1 24.8557,E2 244.1645} C_DIS
LIN {X -118.4305,Y -54.3312,Z 146,A -159.0453,B 24.9626,C -1.4136,E1 24.8541,E2 245.5371} C_DIS
LIN {X -119.767,Y -51.3183,Z 146,A -160.5201,B 24.9624,C -1.4167,E1 24.8524,E2 247.0127} C_DIS
LIN {X -120.9635,Y -48.4298,Z 146,A -161.8519,B 24.9621,C -1.4228,E1 24.851,E2 248.3374} C_DIS
LIN {X -122.0195,Y -45.703,Z 146,A -163.1909,B 24.9621,C -1.4241,E1 24.8497,E2 249.6808} C_DIS
LIN {X -123.1093,Y -42.6806,Z 146,A -164.611,B 24.9618,C -1.4281,E1 24.8484,E2 251.0995} C_DIS
LIN {X -124.1186,Y -39.6499,Z 146,A -166.023,B 24.9616,C -1.432,E1 24.8471,E2 252.5102} C_DIS
LIN {X -125.0612,Y -36.5683,Z 146,A -167.4582,B 24.9614,C -1.4356,E1 24.846,E2 253.9453} C_DIS
LIN {X -125.9375,Y -33.4265,Z 146,A -168.9092,B 24.9612,C -1.4393,E1 24.8449,E2 255.3958} C_DIS
LIN {X -126.8493,Y -29.7896,Z 146,A -170.691,B 24.9612,C -1.4382,E1 24.8437,E2 257.1907} C_DIS
LIN {X -127.6528,Y -26.1219,Z 146,A -172.2089,B 24.9606,C -1.4497,E1 24.8429,E2 258.69} C_DIS
LIN {X -128.2461,Y -23.033,Z 146,A -173.6132,B 24.9604,C -1.4531,E1 24.8422,E2 260.0944} C_DIS
LIN {X -128.7638,Y -19.937,Z 146,A -174.984,B 24.9602,C -1.458,E1 24.8415,E2 261.4619} C_DIS
LIN {X -129.2081,Y -16.8192,Z 146,A -176.4147,B 24.96,C -1.4604,E1 24.841,E2 262.8955} C_DIS
LIN {X -129.6631,Y -12.8559,Z 146,A -178.2243,B 24.9599,C -1.4635,E1 24.8405,E2 264.7086} C_DIS
LIN {X -129.9524,Y -9.4871,Z 146,A -179.6456,B 24.9594,C -1.4714,E1 24.8402,E2 266.1194} C_DIS
LIN {X -130.1527,Y -6.1697,Z 146,A 178.7621,B 24.9595,C -1.4701,E1 24.8399,E2 267.7245} C_DIS
LIN {X -130.2803,Y -2.1677,Z 146,A 177.103,B 24.9589,C -1.4806,E1 24.8398,E2 269.3685} C_DIS
LIN {X -130.2803,Y 2.1677,Z 146,A 175.2056,B 24.9586,C -1.4873,E1 24.8398,E2 271.2613} C_DIS
LIN {X -130.1993,Y 5.0784,Z 146,A 173.9137,B 24.9584,C -1.491,E1 24.8399,E2 272.5523} C_DIS
LIN {X -130.0517,Y 8.0122,Z 146,A 172.6103,B 24.9581,C -1.4947,E1 24.8401,E2 273.8547} C_DIS
LIN {X -129.8395,Y 10.9242,Z 146,A 171.2902,B 24.9581,C -1.4972,E1 24.8404,E2 275.1766} C_DIS
LIN {X -129.5073,Y 14.3404,Z 146,A 169.6442,B 24.9581,C -1.4959,E1 24.8409,E2 276.8358} C_DIS
LIN {X -129.0071,Y 18.2975,Z 146,A 167.9935,B 24.9575,C -1.5064,E1 24.8415,E2 278.4711} C_DIS
LIN {X -128.4969,Y 21.5906,Z 146,A 166.516,B 24.9572,C -1.5107,E1 24.8422,E2 279.9473} C_DIS
LIN {X -127.9073,Y 24.8486,Z 146,A 165.0923,B 24.9569,C -1.5169,E1 24.8429,E2 281.3645} C_DIS
LIN {X -127.1998,Y 28.256,Z 146,A 163.5334,B 24.9567,C -1.5206,E1 24.8438,E2 282.9239} C_DIS
LIN {X -126.5919,Y 30.8573,Z 146,A 162.3597,B 24.9565,C -1.5245,E1 24.8446,E2 284.0952} C_DIS
LIN {X -125.7896,Y 33.981,Z 146,A 160.9465,B 24.9562,C -1.5293,E1 24.8456,E2 285.5052} C_DIS
LIN {X -124.9484,Y 36.9537,Z 146,A 159.511,B 24.9562,C -1.5301,E1 24.8467,E2 286.9471} C_DIS
LIN {X -123.9969,Y 40.031,Z 146,A 158.1329,B 24.9558,C -1.5364,E1 24.8478,E2 288.3181} C_DIS
LIN {X -123.0041,Y 42.9841,Z 146,A 156.6956,B 24.9558,C -1.5376,E1 24.8492,E2 289.7606} C_DIS
LIN {X -121.8497,Y 46.1563,Z 146,A 155.222,B 24.9554,C -1.5428,E1 24.8506,E2 291.2302} C_DIS
LIN {X -120.5463,Y 49.4647,Z 146,A 153.6676,B 24.9551,C -1.5481,E1 24.8522,E2 292.7807} C_DIS
LIN {X -119.2749,Y 52.4564,Z 146,A 152.2273,B 24.9549,C -1.552,E1 24.8538,E2 294.2196} C_DIS
LIN {X -117.9228,Y 55.4292,Z 146,A 150.7802,B 24.9546,C -1.5559,E1 24.8555,E2 295.6652} C_DIS
LIN {X -116.6112,Y 58.1347,Z 146,A 149.4486,B 24.9544,C -1.5595,E1 24.8571,E2 296.9954} C_DIS
LIN {X -114.9549,Y 61.3474,Z 146,A 147.7069,B 24.9546,C -1.5572,E1 24.8594,E2 298.752} C_DIS
LIN {X -112.7667,Y 65.2815,Z 146,A 145.7879,B 24.9541,C -1.5659,E1 24.862,E2 300.6603} C_DIS
LIN {X -110.4985,Y 69.0518,Z 146,A 143.8031,B 24.9539,C -1.5692,E1 24.8649,E2 302.6475} C_DIS
LIN {X -108.1381,Y 72.6934,Z 146,A 141.8851,B 24.9536,C -1.5742,E1 24.8679,E2 304.5632} C_DIS
LIN {X -105.8163,Y 76.033,Z 146,A 140.101,B 24.9533,C -1.5794,E1 24.8707,E2 306.3435} C_DIS
LIN {X -103.2441,Y 79.4911,Z 146,A 138.1773,B 24.953,C -1.5833,E1 24.874,E2 308.2673} C_DIS
LIN {X -100.6268,Y 82.7794,Z 146,A 136.3179,B 24.9528,C -1.5877,E1 24.8772,E2 310.1248} C_DIS
LIN {X -97.9977,Y 85.875,Z 146,A 134.5264,B 24.9525,C -1.5921,E1 24.8805,E2 311.9139} C_DIS
LIN {X -95.0881,Y 89.0865,Z 146,A 132.6018,B 24.9523,C -1.5961,E1 24.8841,E2 313.8374} C_DIS
LIN {X -92.1363,Y 92.1363,Z 146,A 130.7671,B 24.9519,C -1.6022,E1 24.8877,E2 315.6654} C_DIS
LIN {X -89.1255,Y 95.0516,Z 146,A 128.935,B 24.9516,C -1.6072,E1 24.8914,E2 317.4933} C_DIS
LIN {X -86.0603,Y 97.8352,Z 146,A 127.0857,B 24.9514,C -1.6101,E1 24.8953,E2 319.343} C_DIS
LIN {X -82.7794,Y 100.6268,Z 146,A 125.1443,B 24.9513,C -1.6122,E1 24.8994,E2 321.287} C_DIS
LIN {X -79.5093,Y 103.23,Z 146,A 123.3017,B 24.9511,C -1.616,E1 24.9035,E2 323.1273} C_DIS
LIN {X -76.1271,Y 105.7489,Z 146,A 121.4375,B 24.9509,C -1.6194,E1 24.9077,E2 324.9899} C_DIS
LIN {X -72.6934,Y 108.1381,Z 146,A 119.5907,B 24.9507,C -1.6228,E1 24.9119,E2 326.8349} C_DIS
LIN {X -69.1957,Y 110.409,Z 146,A 117.7089,B 24.9506,C -1.624,E1 24.9164,E2 328.7197} C_DIS
LIN {X -65.3985,Y 112.699,Z 146,A 115.8141,B 24.9502,C -1.6303,E1 24.9209,E2 330.6054} C_DIS
LIN {X -61.6694,Y 114.7819,Z 146,A 113.9441,B 24.95,C -1.634,E1 24.9255,E2 332.4719} C_DIS
LIN {X -58.8431,Y 116.2544,Z 146,A 112.5941,B 24.9497,C -1.6388,E1 24.9288,E2 333.8141} C_DIS
LIN {X -55.7328,Y 117.7777,Z 146,A 111.082,B 24.9495,C -1.6418,E1 24.9326,E2 335.3231} C_DIS
LIN {X -52.4564,Y 119.2749,Z 146,A 109.4897,B 24.9494,C -1.6438,E1 24.9366,E2 336.9145} C_DIS
LIN {X -50.0308,Y 120.3099,Z 146,A 108.3306,B 24.9493,C -1.6455,E1 24.9396,E2 338.0721} C_DIS
LIN {X -47.2104,Y 121.4442,Z 146,A 106.9889,B 24.9492,C -1.6472,E1 24.9431,E2 339.4129} C_DIS
LIN {X -44.1935,Y 122.5743,Z 146,A 105.5699,B 24.9491,C -1.6489,E1 24.9468,E2 340.8305} C_DIS
Enddeposition()
END
